      rq_activate_all_grippers(True)
      # end: URCap Program Node
      # begin: URCap Program Node
      #   Source: Robotiq_Grippers, 1.8.13.22852, Robotiq Inc.
      #   Type: Greifer
      $ 271 "Greifer geschlossen (1)"
      if not(gripper_connected[0]):
        popup("Greifer 1 muss verbunden sein, um dieses Programm auszuführen.", "Keine Verbindung", False, True, True)
      end
      if not(rq_is_gripper_activated("1")):
        popup("Greifer 1 ist nicht aktiviert. Wechseln Sie zur Registerkarte Installation > Greifer, um ihn zu aktivieren und das Programm erneut auszuführen.", "Nicht aktiviert", False, True, True)
      end
      rq_set_pos_spd_for(255, 255, 255, "1")
      rq_wait_pos_spe_for_request(255, 255, 255, "1")
      rq_go_to("1")
      rq_wait("1")
      # end: URCap Program Node
      $ 272 "init_qMast≔ False "
      global init_qMast=  False
      $ 273 "Aufruf UserPopups"
      UserPopups()
      $ 274 "Aufruf MachineInputPopUps"
      MachineInputPopUps()
      $ 275 "start_ping≔ True "
      global start_ping=  True
    end
    $ 277 "Switch jobID"
    switch_1 = jobID
    $ 278 "Case 11"
    if (11 == switch_1):
      $ 279 "dest_jobID≔jobArr[1]"
      global dest_jobID=jobArr[1]
      $ 280 "src_dest_p≔qMast.get_loc()"
      global src_dest_p=qMast.get_loc()
      $ 281 "source_p≔src_dest_p[0]"
      global source_p=src_dest_p[0]
      # begin: URCap Program Node
      #   Source: Robotiq_Grippers, 1.8.13.22852, Robotiq Inc.
      #   Type: Greifer
      $ 282 "Greifer geschlossen (1)"
      if not(gripper_connected[0]):
        popup("Greifer 1 muss verbunden sein, um dieses Programm auszuführen.", "Keine Verbindung", False, True, True)
      end
      if not(rq_is_gripper_activated("1")):
        popup("Greifer 1 ist nicht aktiviert. Wechseln Sie zur Registerkarte Installation > Greifer, um ihn zu aktivieren und das Programm erneut auszuführen.", "Nicht aktiviert", False, True, True)
      end
      rq_set_pos_spd_for(255, 255, 255, "1")
      rq_wait_pos_spe_for_request(255, 255, 255, "1")
      rq_go_to("1")
      rq_wait("1")
      # end: URCap Program Node
      $ 283 "FahreAchse"
      $ 284 "stn1_home_p" "breakAfter"
      set_tcp(p[-3.0E-4,2.5E-4,0.1575,0.0,0.0,0.0])
      movej(get_inverse_kin(pose_trans(stn1_plane, pose_trans(p[.053539610991, -.984987293150, -.024848236577, .000189536594, .000276418508, 3.136265531618], stn1_home_p_p)), qnear=stn1_home_p_q), a=3.490658503988659, v=1.0471975511965976, r=0.1)
      $ 285 "FahreAchse"
      $ 286 "stn1_help2_p" "breakAfter"
      set_tcp(p[-3.0E-4,2.5E-4,0.1575,0.0,0.0,0.0])
      movej(get_inverse_kin(pose_trans(stn1_plane, pose_trans(p[.053539610991, -.984987293150, -.024848236577, .000189536594, .000276418508, 3.136265531618], stn1_help2_p_p)), qnear=stn1_help2_p_q), a=1.0471975511965976, v=0.5235987755982988, r=0.05)
      $ 287 "stn1_help_p" "breakAfter"
      set_tcp(p[-3.0E-4,2.5E-4,0.1575,0.0,0.0,0.0])
      movej(get_inverse_kin(pose_trans(stn1_plane, pose_trans(p[.053539610991, -.984987293150, -.024848236577, .000189536594, .000276418508, 3.136265531618], stn1_help_p_p)), qnear=stn1_help_p_q), a=1.0471975511965976, v=0.5235987755982988)
      $ 288 "isStn1Good≔qMast.is_stn1_good()"
      global isStn1Good=qMast.is_stn1_good()
      $ 289 "If isStn1Good ≟  True "
      if (isStn1Good  ==    True  ):
        $ 290 "FahreAchse"
        $ 291 "source_p" "breakAfter"
        set_tcp(p[-3.0E-4,2.5E-4,0.1575,0.0,0.0,0.0])
        movej(pose_trans(stn1_plane, source_p), a=0.8726646259971648, v=0.5235987755982988)
        $ 292 "isStn1Good≔qMast.is_stn1_good()"
        global isStn1Good=qMast.is_stn1_good()
        $ 293 "If isStn1Good ≟  True "
        if (isStn1Good  ==    True  ):
          # begin: URCap Program Node
          #   Source: Robotiq_Grippers, 1.8.13.22852, Robotiq Inc.
          #   Type: Greifer
          $ 294 "Greiferbewegung50% (1)"
          if not(gripper_connected[0]):
            popup("Greifer 1 muss verbunden sein, um dieses Programm auszuführen.", "Keine Verbindung", False, True, True)
          end
          if not(rq_is_gripper_activated("1")):
            popup("Greifer 1 ist nicht aktiviert. Wechseln Sie zur Registerkarte Installation > Greifer, um ihn zu aktivieren und das Programm erneut auszuführen.", "Nicht aktiviert", False, True, True)
          end
          rq_set_pos_spd_for(128, 255, 128, "1")
          rq_wait_pos_spe_for_request(128, 255, 128, "1")
          rq_go_to("1")
          rq_wait("1")
          # end: URCap Program Node
          $ 295 "cur_pose≔pose_trans(pose_inv(stn1_plane), get_actual_tcp_pose())"
          global cur_pose= pose_trans ( pose_inv (stn1_plane),  get_actual_tcp_pose ())
          $ 296 "stn1_pick_p≔pose_trans(cur_pose, p[0,0,stn1_pick_z/1000,0,0,0])"
          global stn1_pick_p= pose_trans (cur_pose, p[0,0,stn1_pick_z/1000,0,0,0])
          $ 297 "FahreLinear"
          $ 298 "stn1_pick_p" "breakAfter"
          set_tcp(p[-3.0E-4,2.5E-4,0.1575,0.0,0.0,0.0])
          movel(pose_trans(stn1_plane, stn1_pick_p), a=0.15, v=0.075)
          $ 299 "isStn1Good≔qMast.is_stn1_good()"
          global isStn1Good=qMast.is_stn1_good()
          $ 300 "If isStn1Good ≟  True "
          if (isStn1Good  ==    True  ):
            # begin: URCap Program Node
            #   Source: Robotiq_Grippers, 1.8.13.22852, Robotiq Inc.
            #   Type: Greifer
            $ 301 "Greifer geschlossen (1)"
            if not(gripper_connected[0]):
              popup("Greifer 1 muss verbunden sein, um dieses Programm auszuführen.", "Keine Verbindung", False, True, True)
            end
            if not(rq_is_gripper_activated("1")):
              popup("Greifer 1 ist nicht aktiviert. Wechseln Sie zur Registerkarte Installation > Greifer, um ihn zu aktivieren und das Programm erneut auszuführen.", "Nicht aktiviert", False, True, True)
            end
            rq_set_pos_spd_for(255, 128, 128, "1")
            rq_wait_pos_spe_for_request(255, 128, 128, "1")
            rq_go_to("1")
            rq_wait("1")
            # end: URCap Program Node
            $ 302 "Warten: 0.2"
            sleep(0.2)
          else:
            $ 303 "Else" "noBreak"
            $ 304 "dest_jobID≔1000"
            global dest_jobID=1000
          end
          $ 305 "FahreAchse"
          $ 306 "source_p" "breakAfter"
          set_tcp(p[-3.0E-4,2.5E-4,0.1575,0.0,0.0,0.0])
          movej(pose_trans(stn1_plane, source_p), a=0.8726646259971648, v=0.5235987755982988)
        else:
          $ 307 "Else" "noBreak"
          $ 308 "dest_jobID≔1000"
          global dest_jobID=1000
        end
      else:
        $ 309 "Else" "noBreak"
        $ 310 "dest_jobID≔1000"
        global dest_jobID=1000
      end
      $ 311 "FahreAchse"
      $ 312 "stn1_help_p" "breakAfter"
      set_tcp(p[-3.0E-4,2.5E-4,0.1575,0.0,0.0,0.0])
      movej(get_inverse_kin(pose_trans(stn1_plane, pose_trans(p[.053539610991, -.984987293150, -.024848236577, .000189536594, .000276418508, 3.136265531618], stn1_help_p_p)), qnear=stn1_help_p_q), a=0.8726646259971648, v=0.5235987755982988, r=0.005)
      $ 313 "stn1_help2_p" "breakAfter"
      set_tcp(p[-3.0E-4,2.5E-4,0.1575,0.0,0.0,0.0])
      movej(get_inverse_kin(pose_trans(stn1_plane, pose_trans(p[.053539610991, -.984987293150, -.024848236577, .000189536594, .000276418508, 3.136265531618], stn1_help2_p_p)), qnear=stn1_help2_p_q), a=0.8726646259971648, v=0.5235987755982988)
      # begin: URCap Program Node
      #   Source: Robotiq_Grippers, 1.8.13.22852, Robotiq Inc.
      #   Type: Griffkontrolle
      $ 314 "Griffkontrolle"
      # begin: URCap Program Node
      #   Source: Robotiq_Grippers, 1.8.13.22852, Robotiq Inc.
      #   Type: Wenn
      $ 315 "Wenn Objekt nicht erkannt          " "noBreak"
      if (not rq_is_object_detected(1)):
        $ 316 "dest_jobID≔1000" "noBreak"
        global dest_jobID=1000
        # end: URCap Program Node
      end
      # end: URCap Program Node
      $ 317 "Switch dest_jobID"
      switch_2 = dest_jobID
      $ 318 "Case 41"
      if (41 == switch_2):
        $ 319 "FahreAchse"
        $ 320 "stn1_home_p" "breakAfter"
        set_tcp(p[-3.0E-4,2.5E-4,0.1575,0.0,0.0,0.0])
        movej(get_inverse_kin(pose_trans(stn1_plane, pose_trans(p[.053539610991, -.984987293150, -.024848236577, .000189536594, .000276418508, 3.136265531618], stn1_home_p_p)), qnear=stn1_home_p_q), a=1.3962634015954636, v=1.0471975511965976, r=0.05)
        $ 321 "FahreAchse"
        $ 322 "stn6_home_p" "breakAfter"
        set_tcp(p[-3.0E-4,2.5E-4,0.1575,0.0,0.0,0.0])
        movej(get_inverse_kin(pose_trans(stn6_plane, pose_trans(p[.776557109756, -.878329076792, .250244777977, -.001605684562, .009314448336, 1.565629725105], stn6_home_p_p)), qnear=stn6_home_p_q), a=3.490658503988659, v=1.0471975511965976, r=0.05)
        $ 323 "stn9_dcap_apr_p" "breakAfter"
        set_tcp(p[-3.0E-4,2.5E-4,0.1575,0.0,0.0,0.0])
        movej(get_inverse_kin(pose_trans(stn6_plane, pose_trans(p[.776557109756, -.878329076792, .250244777977, -.001605684562, .009314448336, 1.565629725105], stn9_dcap_apr_p_p)), qnear=stn9_dcap_apr_p_q), a=3.490658503988659, v=1.0471975511965976)
        $ 324 "Einstellen Decap=Ein"
        set_standard_digital_out(2, True)
        $ 325 "FahreLinear"
        $ 326 "stn9_lv_tb_p" "breakAfter"
        set_tcp(p[-3.0E-4,2.5E-4,0.1575,0.0,0.0,0.0])
        movel(pose_trans(stn6_plane, pose_trans(p[.776557109756, -.878329076792, .250244777977, -.001605684562, .009314448336, 1.565629725105], stn9_lv_tb_p_p)), a=1.2, v=0.25)
        # begin: URCap Program Node
        #   Source: Robotiq_Grippers, 1.8.13.22852, Robotiq Inc.
        #   Type: Greifer
        $ 327 "Greiferbewegung65% (1)"
        if not(gripper_connected[0]):
          popup("Greifer 1 muss verbunden sein, um dieses Programm auszuführen.", "Keine Verbindung", False, True, True)
        end
        if not(rq_is_gripper_activated("1")):
          popup("Greifer 1 ist nicht aktiviert. Wechseln Sie zur Registerkarte Installation > Greifer, um ihn zu aktivieren und das Programm erneut auszuführen.", "Nicht aktiviert", False, True, True)
        end
        rq_set_pos_spd_for(166, 128, 0, "1")
        rq_wait_pos_spe_for_request(166, 128, 0, "1")
        rq_go_to("1")
        rq_wait("1")
        # end: URCap Program Node
        $ 328 "Warten: 0.5"
        sleep(0.5)
        $ 329 "Einstellen Decap=Aus"
        set_standard_digital_out(2, False)
        $ 330 "FahreLinear"
        $ 331 "stn9_hold_cap_p" "breakAfter"
        set_tcp(p[-3.0E-4,2.5E-4,0.1575,0.0,0.0,0.0])
        movel(pose_trans(stn6_plane, pose_trans(p[.776557109756, -.878329076792, .250244777977, -.001605684562, .009314448336, 1.565629725105], stn9_hold_cap_p_p)), a=1.2, v=0.25)
        # begin: URCap Program Node
        #   Source: Robotiq_Grippers, 1.8.13.22852, Robotiq Inc.
        #   Type: Greifer
        $ 332 "Greifer geschlossen (1)"
        if not(gripper_connected[0]):
          popup("Greifer 1 muss verbunden sein, um dieses Programm auszuführen.", "Keine Verbindung", False, True, True)
        end
        if not(rq_is_gripper_activated("1")):
          popup("Greifer 1 ist nicht aktiviert. Wechseln Sie zur Registerkarte Installation > Greifer, um ihn zu aktivieren und das Programm erneut auszuführen.", "Nicht aktiviert", False, True, True)
        end
        rq_set_pos_spd_for(255, 128, 128, "1")
        rq_wait_pos_spe_for_request(255, 128, 128, "1")
        rq_go_to("1")
        rq_wait("1")
        # end: URCap Program Node
        $ 333 "Einstellen Decap=Ein"
        set_standard_digital_out(2, True)
        $ 334 "FahreLinear"
        $ 335 "stn9_dcap_apr_p" "breakAfter"
        set_tcp(p[-3.0E-4,2.5E-4,0.1575,0.0,0.0,0.0])
        movel(pose_trans(stn6_plane, pose_trans(p[.776557109756, -.878329076792, .250244777977, -.001605684562, .009314448336, 1.565629725105], stn9_dcap_apr_p_p)), a=1.2, v=0.25)
        $ 336 "Aufruf stn4_grab_loop"
        stn4_grab_loop()
        $ 337 "dest2_jobID≔qMast.stn4_get_next(stn4_tube_ok)"
        global dest2_jobID=qMast.stn4_get_next(stn4_tube_ok)
        $ 338 "src_dest_p≔qMast.get_loc()"
        global src_dest_p=qMast.get_loc()
        $ 339 "dest_p≔src_dest_p[0]"
        global dest_p=src_dest_p[0]
        $ 340 "Switch dest2_jobID"
        switch_3 = dest2_jobID
        $ 341 "Case 52"
        if (52 == switch_3):
          $ 342 "FahreAchse"
          $ 343 "stn5_stn4_hlp_p" "breakAfter"
          set_tcp(p[-3.0E-4,2.5E-4,0.1575,0.0,0.0,0.0])
          movej(get_inverse_kin(pose_trans(stn6_plane, pose_trans(p[.776557109756, -.878329076792, .250244777977, -.001605684562, .009314448336, 1.565629725105], stn5_stn4_hlp_p_p)), qnear=stn5_stn4_hlp_p_q), a=3.490658503988659, v=1.0471975511965976, r=0.05)
          $ 344 "FahreLinear"
          $ 345 "dest_p" "breakAfter"
          set_tcp(p[-3.0E-4,2.5E-4,0.1575,0.0,0.0,0.0])
          movel(pose_trans(stn5_plane, dest_p), a=1.2, v=0.5)
          $ 346 "cur_pose≔pose_trans(pose_inv(stn5_plane), get_actual_tcp_pose())"
          global cur_pose= pose_trans ( pose_inv (stn5_plane),  get_actual_tcp_pose ())
          $ 347 "stn5_place_z_p≔pose_trans(cur_pose, p[0,0,stn5_place_tb_z/1000,0,0,0])"
          global stn5_place_z_p= pose_trans (cur_pose, p[0,0,stn5_place_tb_z/1000,0,0,0])
          $ 348 "FahreLinear"
          $ 349 "stn5_place_z_p" "breakAfter"
          set_tcp(p[-3.0E-4,2.5E-4,0.1575,0.0,0.0,0.0])
          movel(pose_trans(stn5_plane, stn5_place_z_p), a=0.5, v=0.1)
          # begin: URCap Program Node
          #   Source: Robotiq_Grippers, 1.8.13.22852, Robotiq Inc.
          #   Type: Greifer
          $ 350 "Greiferbewegung50% (1)"
          if not(gripper_connected[0]):
            popup("Greifer 1 muss verbunden sein, um dieses Programm auszuführen.", "Keine Verbindung", False, True, True)
          end
          if not(rq_is_gripper_activated("1")):
            popup("Greifer 1 ist nicht aktiviert. Wechseln Sie zur Registerkarte Installation > Greifer, um ihn zu aktivieren und das Programm erneut auszuführen.", "Nicht aktiviert", False, True, True)
          end
          rq_set_pos_spd_for(127, 255, 255, "1")
          rq_wait_pos_spe_for_request(127, 255, 255, "1")
          rq_go_to("1")
          rq_wait("1")
          # end: URCap Program Node
          $ 351 "dest_p" "breakAfter"
          set_tcp(p[-3.0E-4,2.5E-4,0.1575,0.0,0.0,0.0])
          movel(pose_trans(stn5_plane, dest_p), a=1.2, v=0.25)
          # begin: URCap Program Node
          #   Source: Robotiq_Grippers, 1.8.13.22852, Robotiq Inc.
          #   Type: Greifer
          $ 352 "Greifer geschlossen (1)"
          if not(gripper_connected[0]):
            popup("Greifer 1 muss verbunden sein, um dieses Programm auszuführen.", "Keine Verbindung", False, True, True)
          end
          if not(rq_is_gripper_activated("1")):
            popup("Greifer 1 ist nicht aktiviert. Wechseln Sie zur Registerkarte Installation > Greifer, um ihn zu aktivieren und das Programm erneut auszuführen.", "Nicht aktiviert", False, True, True)
          end
          rq_set_pos_spd_for(255, 255, 255, "1")
          rq_wait_pos_spe_for_request(255, 255, 255, "1")
          rq_go_to("1")
          rq_wait("1")
          # end: URCap Program Node
          $ 353 "FahreAchse"
          $ 354 "stn5_stn4_hlp_p" "breakAfter"
          set_tcp(p[-3.0E-4,2.5E-4,0.1575,0.0,0.0,0.0])
          movej(get_inverse_kin(pose_trans(stn6_plane, pose_trans(p[.776557109756, -.878329076792, .250244777977, -.001605684562, .009314448336, 1.565629725105], stn5_stn4_hlp_p_p)), qnear=stn5_stn4_hlp_p_q), a=1.3962634015954636, v=1.0471975511965976, r=0.05)
          $ 355 "stn6_home_p" "breakAfter"
          set_tcp(p[-3.0E-4,2.5E-4,0.1575,0.0,0.0,0.0])
          movej(get_inverse_kin(pose_trans(stn6_plane, pose_trans(p[.776557109756, -.878329076792, .250244777977, -.001605684562, .009314448336, 1.565629725105], stn6_home_p_p)), qnear=stn6_home_p_q), a=1.3962634015954636, v=1.0471975511965976)
          $ 356 "Aufruf reset_jobs"
          reset_jobs()
        elif (72 == switch_3):
          $ 357 "Case 72"
          $ 358 "FahreAchse"
          $ 359 "stn6_home_p" "breakAfter"
          set_tcp(p[-3.0E-4,2.5E-4,0.1575,0.0,0.0,0.0])
          movej(get_inverse_kin(pose_trans(stn6_plane, pose_trans(p[.776557109756, -.878329076792, .250244777977, -.001605684562, .009314448336, 1.565629725105], stn6_home_p_p)), qnear=stn6_home_p_q), a=3.490658503988659, v=1.0471975511965976, r=0.1)
          $ 360 "FahreAchse"
          $ 361 "stn7_home_p" "breakAfter"
          set_tcp(p[-3.0E-4,2.5E-4,0.1575,0.0,0.0,0.0])
          movej(get_inverse_kin(pose_trans(stn7_plane, pose_trans(p[.109811488584, -1.023382701287, -.166619380160, .003048702642, -.008599620441, 2.442192581404], stn7_home_p_p)), qnear=stn7_home_p_q), a=3.490658503988659, v=1.0471975511965976, r=0.1)
          $ 362 "Aufruf stn7_check_doors"
          stn7_check_doors()
          $ 363 "FahreAchse"
          $ 364 "dest_p" "breakAfter"
          set_tcp(p[-3.0E-4,2.5E-4,0.1575,0.0,0.0,0.0])
          movej(pose_trans(stn7_plane, dest_p), a=3.490658503988659, v=1.0471975511965976)
          $ 365 "cur_pose≔pose_trans(pose_inv(stn7_plane), get_actual_tcp_pose())"
          global cur_pose= pose_trans ( pose_inv (stn7_plane),  get_actual_tcp_pose ())
          $ 366 "stn7_place_p≔pose_trans(cur_pose, p[0,0,stn7_place_z/1000,0,0,0])"
          global stn7_place_p= pose_trans (cur_pose, p[0,0,stn7_place_z/1000,0,0,0])
          $ 367 "FahreLinear"
          $ 368 "stn7_place_p" "breakAfter"
          set_tcp(p[-3.0E-4,2.5E-4,0.1575,0.0,0.0,0.0])
          movel(pose_trans(stn7_plane, stn7_place_p), a=0.15, v=0.075)
          # begin: URCap Program Node
          #   Source: Robotiq_Grippers, 1.8.13.22852, Robotiq Inc.
          #   Type: Greifer
          $ 369 "Greifer offen (1)"
          if not(gripper_connected[0]):
            popup("Greifer 1 muss verbunden sein, um dieses Programm auszuführen.", "Keine Verbindung", False, True, True)
          end
          if not(rq_is_gripper_activated("1")):
            popup("Greifer 1 ist nicht aktiviert. Wechseln Sie zur Registerkarte Installation > Greifer, um ihn zu aktivieren und das Programm erneut auszuführen.", "Nicht aktiviert", False, True, True)
          end
          rq_set_pos_spd_for(0, 255, 255, "1")
          rq_wait_pos_spe_for_request(0, 255, 255, "1")
          rq_go_to("1")
          rq_wait("1")
          # end: URCap Program Node
          $ 370 "FahreLinear"
          $ 371 "dest_p" "breakAfter"
          set_tcp(p[-3.0E-4,2.5E-4,0.1575,0.0,0.0,0.0])
          movel(pose_trans(stn7_plane, dest_p), a=1.2, v=0.25)
          # begin: URCap Program Node
          #   Source: Robotiq_Grippers, 1.8.13.22852, Robotiq Inc.
          #   Type: Greifer
          $ 372 "Greifer geschlossen (1)"
          if not(gripper_connected[0]):
            popup("Greifer 1 muss verbunden sein, um dieses Programm auszuführen.", "Keine Verbindung", False, True, True)
          end
          if not(rq_is_gripper_activated("1")):
            popup("Greifer 1 ist nicht aktiviert. Wechseln Sie zur Registerkarte Installation > Greifer, um ihn zu aktivieren und das Programm erneut auszuführen.", "Nicht aktiviert", False, True, True)
          end
          rq_set_pos_spd_for(255, 255, 255, "1")
          rq_wait_pos_spe_for_request(255, 255, 255, "1")
          rq_go_to("1")
          rq_wait("1")
          # end: URCap Program Node
          $ 373 "FahreAchse"
          $ 374 "stn7_home_p" "breakAfter"
          set_tcp(p[-3.0E-4,2.5E-4,0.1575,0.0,0.0,0.0])
          movej(get_inverse_kin(pose_trans(stn7_plane, pose_trans(p[.109811488584, -1.023382701287, -.166619380160, .003048702642, -.008599620441, 2.442192581404], stn7_home_p_p)), qnear=stn7_home_p_q), a=3.490658503988659, v=1.0471975511965976)
          $ 375 "Aufruf reset_jobs"
          reset_jobs()
        elif (102 == switch_3):
          $ 376 "Case 102"
          $ 377 "FahreAchse"
          $ 378 "stn6_home_p" "breakAfter"
          set_tcp(p[-3.0E-4,2.5E-4,0.1575,0.0,0.0,0.0])
          movej(get_inverse_kin(pose_trans(stn6_plane, pose_trans(p[.776557109756, -.878329076792, .250244777977, -.001605684562, .009314448336, 1.565629725105], stn6_home_p_p)), qnear=stn6_home_p_q), a=3.490658503988659, v=1.0471975511965976, r=0.1)
          $ 379 "stn10_hlp_p" "breakAfter"
          set_tcp(p[-3.0E-4,2.5E-4,0.1575,0.0,0.0,0.0])
          movej(get_inverse_kin(pose_trans(stn6_plane, pose_trans(p[.779413821965, -.869656427631, .149271774994, -.000554336510, .003016566406, 1.568064465904], stn10_hlp_p_p)), qnear=stn10_hlp_p_q), a=3.490658503988659, v=1.0471975511965976)
          $ 380 "FahreLinear"
          $ 381 "dest_p" "breakAfter"
          set_tcp(p[-3.0E-4,2.5E-4,0.1575,0.0,0.0,0.0])
          movel(pose_trans(stn6_plane, dest_p), a=1.2, v=0.5)
          $ 382 "cur_pose≔pose_trans(pose_inv(stn6_plane), get_actual_tcp_pose())"
          global cur_pose= pose_trans ( pose_inv (stn6_plane),  get_actual_tcp_pose ())
          $ 384 "stn10_place_p≔pose_trans(cur_pose, p[0,0,stn10_place_z/1000,0,0,0])"
          global stn10_place_p= pose_trans (cur_pose, p[0,0,stn10_place_z/1000,0,0,0])
          $ 385 "FahreLinear"
          $ 386 "stn10_place_p" "breakAfter"
          set_tcp(p[-3.0E-4,2.5E-4,0.1575,0.0,0.0,0.0])
          movel(pose_trans(stn6_plane, stn10_place_p), a=1.2, v=0.05)
          # begin: URCap Program Node
          #   Source: Robotiq_Grippers, 1.8.13.22852, Robotiq Inc.
          #   Type: Greifer
          $ 387 "Greiferbewegung50% (1)"
          if not(gripper_connected[0]):
            popup("Greifer 1 muss verbunden sein, um dieses Programm auszuführen.", "Keine Verbindung", False, True, True)
          end
          if not(rq_is_gripper_activated("1")):
            popup("Greifer 1 ist nicht aktiviert. Wechseln Sie zur Registerkarte Installation > Greifer, um ihn zu aktivieren und das Programm erneut auszuführen.", "Nicht aktiviert", False, True, True)
          end
          rq_set_pos_spd_for(127, 255, 0, "1")
          rq_wait_pos_spe_for_request(127, 255, 0, "1")
          rq_go_to("1")
          rq_wait("1")
          # end: URCap Program Node
          $ 388 "dest_p" "breakAfter"
          set_tcp(p[-3.0E-4,2.5E-4,0.1575,0.0,0.0,0.0])
          movel(pose_trans(stn6_plane, dest_p), a=1.2, v=0.25)
          # begin: URCap Program Node
          #   Source: Robotiq_Grippers, 1.8.13.22852, Robotiq Inc.
          #   Type: Greifer
          $ 389 "Greifer geschlossen (1)"
          if not(gripper_connected[0]):
            popup("Greifer 1 muss verbunden sein, um dieses Programm auszuführen.", "Keine Verbindung", False, True, True)
          end
          if not(rq_is_gripper_activated("1")):
            popup("Greifer 1 ist nicht aktiviert. Wechseln Sie zur Registerkarte Installation > Greifer, um ihn zu aktivieren und das Programm erneut auszuführen.", "Nicht aktiviert", False, True, True)
          end
          rq_set_pos_spd_for(255, 255, 255, "1")
          rq_wait_pos_spe_for_request(255, 255, 255, "1")
          rq_go_to("1")
          rq_wait("1")
          # end: URCap Program Node
          $ 390 "FahreAchse"
          $ 391 "stn10_hlp_p" "breakAfter"
          set_tcp(p[-3.0E-4,2.5E-4,0.1575,0.0,0.0,0.0])
          movej(get_inverse_kin(pose_trans(stn6_plane, pose_trans(p[.779413821965, -.869656427631, .149271774994, -.000554336510, .003016566406, 1.568064465904], stn10_hlp_p_p)), qnear=stn10_hlp_p_q), a=3.490658503988659, v=1.0471975511965976, r=0.05)
          $ 392 "stn6_home_p" "breakAfter"
          set_tcp(p[-3.0E-4,2.5E-4,0.1575,0.0,0.0,0.0])
          movej(get_inverse_kin(pose_trans(stn6_plane, pose_trans(p[.776557109756, -.878329076792, .250244777977, -.001605684562, .009314448336, 1.565629725105], stn6_home_p_p)), qnear=stn6_home_p_q), a=3.490658503988659, v=1.0471975511965976)
          $ 393 "Aufruf reset_jobs"
          reset_jobs()
        elif (152 == switch_3):
          $ 394 "Case 152"
          $ 395 "FahreAchse"
          $ 396 "stn11_hlp_p" "breakAfter"
          set_tcp(p[-3.0E-4,2.5E-4,0.1575,0.0,0.0,0.0])
          movej(get_inverse_kin(pose_trans(stn6_plane, pose_trans(p[.776557109756, -.878329076792, .250244777977, -.001605684562, .009314448336, 1.565629725105], stn11_hlp_p_p)), qnear=stn11_hlp_p_q), a=2.0943951023931953, v=1.0471975511965976, r=0.05)
          $ 397 "stn15_home_p" "breakAfter"
          set_tcp(p[-3.0E-4,2.5E-4,0.1575,0.0,0.0,0.0])
          movej(get_inverse_kin(pose_trans(stn6_plane, pose_trans(p[.776557109756, -.878329076792, .250244777977, -.001605684562, .009314448336, 1.565629725105], stn15_home_p_p)), qnear=stn15_home_p_q), a=2.0943951023931953, v=1.0471975511965976, r=0.01)
          $ 398 "dest_p" "breakAfter"
          set_tcp(p[-3.0E-4,2.5E-4,0.1575,0.0,0.0,0.0])
          movej(pose_trans(stn6_plane, dest_p), a=2.0943951023931953, v=1.0471975511965976)
          $ 399 "cur_pose≔pose_trans(pose_inv(stn6_plane), get_actual_tcp_pose())"
          global cur_pose= pose_trans ( pose_inv (stn6_plane),  get_actual_tcp_pose ())
          $ 400 "stn15_place_z_p≔pose_trans(cur_pose, p[0,0,stn15_place_z/1000,0,0,0])"
          global stn15_place_z_p= pose_trans (cur_pose, p[0,0,stn15_place_z/1000,0,0,0])
          $ 401 "FahreLinear"
          $ 402 "stn15_place_z_p" "breakAfter"
          set_tcp(p[-3.0E-4,2.5E-4,0.1575,0.0,0.0,0.0])
          movel(pose_trans(stn6_plane, stn15_place_z_p), a=0.5, v=0.1)
          # begin: URCap Program Node
          #   Source: Robotiq_Grippers, 1.8.13.22852, Robotiq Inc.
          #   Type: Greifer
          $ 403 "Greiferbewegung50% (1)"
          if not(gripper_connected[0]):
            popup("Greifer 1 muss verbunden sein, um dieses Programm auszuführen.", "Keine Verbindung", False, True, True)
          end
          if not(rq_is_gripper_activated("1")):
            popup("Greifer 1 ist nicht aktiviert. Wechseln Sie zur Registerkarte Installation > Greifer, um ihn zu aktivieren und das Programm erneut auszuführen.", "Nicht aktiviert", False, True, True)
          end
          rq_set_pos_spd_for(128, 255, 255, "1")
          rq_wait_pos_spe_for_request(128, 255, 255, "1")
          rq_go_to("1")
          rq_wait("1")
          # end: URCap Program Node
          $ 404 "dest_p" "breakAfter"
          set_tcp(p[-3.0E-4,2.5E-4,0.1575,0.0,0.0,0.0])
          movel(pose_trans(stn6_plane, dest_p), a=0.5, v=0.1)
          # begin: URCap Program Node
          #   Source: Robotiq_Grippers, 1.8.13.22852, Robotiq Inc.
          #   Type: Greifer
          $ 405 "Greifer geschlossen (1)"
          if not(gripper_connected[0]):
            popup("Greifer 1 muss verbunden sein, um dieses Programm auszuführen.", "Keine Verbindung", False, True, True)
          end
          if not(rq_is_gripper_activated("1")):
            popup("Greifer 1 ist nicht aktiviert. Wechseln Sie zur Registerkarte Installation > Greifer, um ihn zu aktivieren und das Programm erneut auszuführen.", "Nicht aktiviert", False, True, True)
          end
          rq_set_pos_spd_for(255, 255, 255, "1")
          rq_wait_pos_spe_for_request(255, 255, 255, "1")
          rq_go_to("1")
          rq_wait("1")
          # end: URCap Program Node
          $ 406 "FahreAchse"
          $ 407 "stn15_home_p" "breakAfter"
          set_tcp(p[-3.0E-4,2.5E-4,0.1575,0.0,0.0,0.0])
          movej(get_inverse_kin(pose_trans(stn6_plane, pose_trans(p[.776557109756, -.878329076792, .250244777977, -.001605684562, .009314448336, 1.565629725105], stn15_home_p_p)), qnear=stn15_home_p_q), a=2.0943951023931953, v=1.0471975511965976, r=0.05)
          $ 408 "FahreAchse"
          $ 409 "stn1_home_p" "breakAfter"
          set_tcp(p[-3.0E-4,2.5E-4,0.1575,0.0,0.0,0.0])
          movej(get_inverse_kin(pose_trans(stn1_plane, pose_trans(p[.053539610991, -.984987293150, -.024848236577, .000189536594, .000276418508, 3.136265531618], stn1_home_p_p)), qnear=stn1_home_p_q), a=2.0943951023931953, v=1.0471975511965976)
          $ 410 "Aufruf reset_jobs"
          reset_jobs()
        end
      elif (1000 == switch_2):
        $ 411 "Case 1000"
        $ 412 "FahreAchse"
        $ 413 "stn1_home_p" "breakAfter"
        set_tcp(p[-3.0E-4,2.5E-4,0.1575,0.0,0.0,0.0])
        movej(get_inverse_kin(pose_trans(stn1_plane, pose_trans(p[.053539610991, -.984987293150, -.024848236577, .000189536594, .000276418508, 3.136265531618], stn1_home_p_p)), qnear=stn1_home_p_q), a=3.490658503988659, v=1.0471975511965976)
        # begin: URCap Program Node
        #   Source: Robotiq_Grippers, 1.8.13.22852, Robotiq Inc.
        #   Type: Greifer
        $ 414 "Greifer geschlossen (1)"
        if not(gripper_connected[0]):
          popup("Greifer 1 muss verbunden sein, um dieses Programm auszuführen.", "Keine Verbindung", False, True, True)
        end
        if not(rq_is_gripper_activated("1")):
          popup("Greifer 1 ist nicht aktiviert. Wechseln Sie zur Registerkarte Installation > Greifer, um ihn zu aktivieren und das Programm erneut auszuführen.", "Nicht aktiviert", False, True, True)
        end
        rq_set_pos_spd_for(255, 128, 128, "1")
        rq_wait_pos_spe_for_request(255, 128, 128, "1")
        rq_go_to("1")
        rq_wait("1")
        # end: URCap Program Node
        $ 415 "Aufruf reset_jobs"
        reset_jobs()
      end
    elif (21 == switch_1):
      $ 416 "Case 21"
      $ 417 "dest_jobID≔jobArr[1]"
      global dest_jobID=jobArr[1]
      $ 418 "src_dest_p≔qMast.get_loc()"
      global src_dest_p=qMast.get_loc()
      $ 419 "source_p≔src_dest_p[0]"
      global source_p=src_dest_p[0]
      $ 420 "Switch dest_jobID"
      switch_2 = dest_jobID
      $ 421 "Case 142"
      if (142 == switch_2):
        $ 422 "FahreAchse"
        $ 423 "stn2_home_p" "breakAfter"
        set_tcp(p[-3.0E-4,2.5E-4,0.1575,0.0,0.0,0.0])
        movej(get_inverse_kin(pose_trans(stn2_plane, pose_trans(p[.137500819741, -.686313800478, .149495066037, -.008721928164, .022313263547, 3.131433712319], stn2_home_p_p)), qnear=stn2_home_p_q), a=1.3962634015954636, v=1.0471975511965976)
        $ 424 "source_p" "breakAfter"
        set_tcp(p[-3.0E-4,2.5E-4,0.1575,0.0,0.0,0.0])
        movej(pose_trans(stn2_plane, source_p), a=1.3962634015954636, v=1.0471975511965976)
        # begin: URCap Program Node
        #   Source: Robotiq_Grippers, 1.8.13.22852, Robotiq Inc.
        #   Type: Greifer
        $ 425 "Greiferbewegung35% (1)"
        if not(gripper_connected[0]):
          popup("Greifer 1 muss verbunden sein, um dieses Programm auszuführen.", "Keine Verbindung", False, True, True)
        end
        if not(rq_is_gripper_activated("1")):
          popup("Greifer 1 ist nicht aktiviert. Wechseln Sie zur Registerkarte Installation > Greifer, um ihn zu aktivieren und das Programm erneut auszuführen.", "Nicht aktiviert", False, True, True)
        end
        rq_set_pos_spd_for(89, 255, 255, "1")
        rq_wait_pos_spe_for_request(89, 255, 255, "1")
        rq_go_to("1")
        rq_wait("1")
        # end: URCap Program Node
        $ 426 "cur_pose≔pose_trans(pose_inv(stn2_plane), get_actual_tcp_pose())"
        global cur_pose= pose_trans ( pose_inv (stn2_plane),  get_actual_tcp_pose ())
        $ 427 "stn2_pick_z_p≔pose_trans(cur_pose, p[0,0,stn2_pk_rk_z/1000,0,0,0])"
        global stn2_pick_z_p= pose_trans (cur_pose, p[0,0,stn2_pk_rk_z/1000,0,0,0])
        $ 428 "FahreLinear"
        $ 429 "stn2_pick_z_p" "breakAfter"
        set_tcp(p[-3.0E-4,2.5E-4,0.1575,0.0,0.0,0.0])
        movel(pose_trans(stn2_plane, stn2_pick_z_p), a=0.5, v=0.1)
        $ 430 "cur_pose≔pose_trans(pose_inv(stn2_plane), get_actual_tcp_pose())"
        global cur_pose= pose_trans ( pose_inv (stn2_plane),  get_actual_tcp_pose ())
        $ 431 "stn2_rk_chk_y_p≔pose_trans(cur_pose, p[0,stn2_rk_chk_y/1000,0,0,0,0])"
        global stn2_rk_chk_y_p= pose_trans (cur_pose, p[0,stn2_rk_chk_y/1000,0,0,0,0])
        $ 432 "FahreLinear"
        $ 433 "stn2_rk_chk_y_p" "breakAfter"
        set_tcp(p[-3.0E-4,2.5E-4,0.1575,0.0,0.0,0.0])
        movel(pose_trans(stn2_plane, stn2_rk_chk_y_p), a=0.5, v=0.1)
        $ 434 "stn14_angle≔0"
        global stn14_angle=0
        $ 435 "stn2_rack_yes≔ False "
        global stn2_rack_yes=  False
        # begin: URCap Program Node
        #   Source: Robotiq_Grippers, 1.8.13.22852, Robotiq Inc.
        #   Type: Greifer
        $ 436 "Greifer geschlossen (1)"
        if not(gripper_connected[0]):
          popup("Greifer 1 muss verbunden sein, um dieses Programm auszuführen.", "Keine Verbindung", False, True, True)
        end
        if not(rq_is_gripper_activated("1")):
          popup("Greifer 1 ist nicht aktiviert. Wechseln Sie zur Registerkarte Installation > Greifer, um ihn zu aktivieren und das Programm erneut auszuführen.", "Nicht aktiviert", False, True, True)
        end
        rq_set_pos_spd_for(255, 0, 0, "1")
        rq_wait_pos_spe_for_request(255, 0, 0, "1")
        rq_go_to("1")
        rq_wait("1")
        # end: URCap Program Node
        $ 437 "gripper_pos≔rq_current_pos_norm()"
        global gripper_pos=rq_current_pos_norm()
        $ 438 "If gripper_pos ≤ 65 and gripper_pos ≥ 57"
        if (gripper_pos  <=  65  and  gripper_pos  >=  57):
          $ 439 "stn2_rack_yes≔ True "
          global stn2_rack_yes=  True
          $ 440 "stn14_angle≔180"
          global stn14_angle=180
        else:
          $ 441 "ElseIf gripper_pos > 65  and gripper_pos ≤ 90"
          if (gripper_pos > 65   and  gripper_pos  <=  90):
            $ 442 "stn2_rack_yes≔ True "
            global stn2_rack_yes=  True
          else:
            $ 443 "Else" "noBreak"
            $ 444 "stn2_rack_yes≔ False "
            global stn2_rack_yes=  False
          end
        end
        # begin: URCap Program Node
        #   Source: Robotiq_Grippers, 1.8.13.22852, Robotiq Inc.
        #   Type: Greifer
        $ 445 "Greiferbewegung35% (1)"
        if not(gripper_connected[0]):
          popup("Greifer 1 muss verbunden sein, um dieses Programm auszuführen.", "Keine Verbindung", False, True, True)
        end
        if not(rq_is_gripper_activated("1")):
          popup("Greifer 1 ist nicht aktiviert. Wechseln Sie zur Registerkarte Installation > Greifer, um ihn zu aktivieren und das Programm erneut auszuführen.", "Nicht aktiviert", False, True, True)
        end
        rq_set_pos_spd_for(89, 255, 255, "1")
        rq_wait_pos_spe_for_request(89, 255, 255, "1")
        rq_go_to("1")
        rq_wait("1")
        # end: URCap Program Node
        $ 446 "FahreLinear"
        $ 447 "stn2_pick_z_p" "breakAfter"
        set_tcp(p[-3.0E-4,2.5E-4,0.1575,0.0,0.0,0.0])
        movel(pose_trans(stn2_plane, stn2_pick_z_p), a=1.2, v=0.25)
        $ 448 "If stn2_rack_yes ≟  True "
        if (stn2_rack_yes  ==    True  ):
          # begin: URCap Program Node
          #   Source: Robotiq_Grippers, 1.8.13.22852, Robotiq Inc.
          #   Type: Greifer
          $ 449 "Greifer geschlossen (1)"
          if not(gripper_connected[0]):
            popup("Greifer 1 muss verbunden sein, um dieses Programm auszuführen.", "Keine Verbindung", False, True, True)
          end
          if not(rq_is_gripper_activated("1")):
            popup("Greifer 1 ist nicht aktiviert. Wechseln Sie zur Registerkarte Installation > Greifer, um ihn zu aktivieren und das Programm erneut auszuführen.", "Nicht aktiviert", False, True, True)
          end
          rq_set_pos_spd_for(255, 128, 255, "1")
          rq_wait_pos_spe_for_request(255, 128, 255, "1")
          rq_go_to("1")
          rq_wait("1")
          # end: URCap Program Node
          $ 450 "FahreLinear"
          $ 451 "source_p" "breakAfter"
          set_tcp(p[-3.0E-4,2.5E-4,0.1575,0.0,0.0,0.0])
          movel(pose_trans(stn2_plane, source_p), a=0.5, v=0.1)
          $ 452 "FahreAchse"
          $ 453 "stn2_home_p" "breakAfter"
          set_tcp(p[-3.0E-4,2.5E-4,0.1575,0.0,0.0,0.0])
          movej(get_inverse_kin(pose_trans(stn2_plane, pose_trans(p[.137500819741, -.686313800478, .149495066037, -.008721928164, .022313263547, 3.131433712319], stn2_home_p_p)), qnear=stn2_home_p_q), a=1.3962634015954636, v=1.0471975511965976)
          $ 454 "FahreAchse"
          $ 455 "stn6_home_p" "breakAfter"
          set_tcp(p[-3.0E-4,2.5E-4,0.1575,0.0,0.0,0.0])
          movej(get_inverse_kin(pose_trans(stn6_plane, pose_trans(p[.776557109756, -.878329076792, .250244777977, -.001605684562, .009314448336, 1.565629725105], stn6_home_p_p)), qnear=stn6_home_p_q), a=1.3962634015954636, v=1.0471975511965976, r=0.1)
          $ 456 "stn14_pl_rk_h_p" "breakAfter"
          set_tcp(p[-3.0E-4,2.5E-4,0.1575,0.0,0.0,0.0])
          movej(get_inverse_kin(pose_trans(stn6_plane, pose_trans(p[.776557109756, -.878329076792, .250244777977, -.001605684562, .009314448336, 1.565629725105], stn14_pl_rk_h_p_p)), qnear=stn14_pl_rk_h_p_q), a=1.3962634015954636, v=1.0471975511965976, r=0.05)
          $ 457 "stn14_pl_rk_p" "breakAfter"
          set_tcp(p[-3.0E-4,2.5E-4,0.1575,0.0,0.0,0.0])
          movej(get_inverse_kin(pose_trans(stn6_plane, pose_trans(p[.776557109756, -.878329076792, .250244777977, -.001605684562, .009314448336, 1.565629725105], stn14_pl_rk_p_p)), qnear=stn14_pl_rk_p_q), a=1.3962634015954636, v=1.0471975511965976)
          $ 458 "If stn14_angle ≟ 180"
          if (stn14_angle  ==  180):
            $ 459 "FahreAchse"
            $ 460 "stn14_plrk_rt_p" "breakAfter"
            set_tcp(p[-3.0E-4,2.5E-4,0.1575,0.0,0.0,0.0])
            movej(get_inverse_kin(pose_trans(stn6_plane, pose_trans(p[.776557109756, -.878329076792, .250244777977, -.001605684562, .009314448336, 1.565629725105], stn14_plrk_rt_p_p)), qnear=stn14_plrk_rt_p_q), a=13.962634015954636, v=3.141592653589793)
            $ 461 "FahreLinear"
            $ 462 "cur_pose≔pose_trans(pose_inv(stn6_plane), get_actual_tcp_pose())"
            global cur_pose= pose_trans ( pose_inv (stn6_plane),  get_actual_tcp_pose ())
            $ 463 "stn14_pl_rk_z_p≔pose_trans(cur_pose, p[0,0,stn14_pl_rk_z/1000,0,0,0])"
            global stn14_pl_rk_z_p= pose_trans (cur_pose, p[0,0,stn14_pl_rk_z/1000,0,0,0])
            $ 464 "stn14_pl_rk_z_p" "breakAfter"
            set_tcp(p[-3.0E-4,2.5E-4,0.1575,0.0,0.0,0.0])
            movel(pose_trans(stn6_plane, stn14_pl_rk_z_p), a=0.5, v=0.05)
            # begin: URCap Program Node
            #   Source: Robotiq_Grippers, 1.8.13.22852, Robotiq Inc.
            #   Type: Greifer
            $ 465 "Greiferbewegung35% (1)"
            if not(gripper_connected[0]):
              popup("Greifer 1 muss verbunden sein, um dieses Programm auszuführen.", "Keine Verbindung", False, True, True)
            end
            if not(rq_is_gripper_activated("1")):
              popup("Greifer 1 ist nicht aktiviert. Wechseln Sie zur Registerkarte Installation > Greifer, um ihn zu aktivieren und das Programm erneut auszuführen.", "Nicht aktiviert", False, True, True)
            end
            rq_set_pos_spd_for(89, 255, 255, "1")
            rq_wait_pos_spe_for_request(89, 255, 255, "1")
            rq_go_to("1")
            rq_wait("1")
            # end: URCap Program Node
            $ 466 "stn14_plrk_rt_p" "breakAfter"
            set_tcp(p[-3.0E-4,2.5E-4,0.1575,0.0,0.0,0.0])
            movel(pose_trans(stn6_plane, pose_trans(p[.776557109756, -.878329076792, .250244777977, -.001605684562, .009314448336, 1.565629725105], stn14_plrk_rt_p_p)), a=0.6, v=0.1)
            # begin: URCap Program Node
            #   Source: Robotiq_Grippers, 1.8.13.22852, Robotiq Inc.
            #   Type: Greifer
            $ 467 "Greifer geschlossen (1)"
            if not(gripper_connected[0]):
              popup("Greifer 1 muss verbunden sein, um dieses Programm auszuführen.", "Keine Verbindung", False, True, True)
            end
            if not(rq_is_gripper_activated("1")):
              popup("Greifer 1 ist nicht aktiviert. Wechseln Sie zur Registerkarte Installation > Greifer, um ihn zu aktivieren und das Programm erneut auszuführen.", "Nicht aktiviert", False, True, True)
            end
            rq_set_pos_spd_for(255, 255, 255, "1")
            rq_wait_pos_spe_for_request(255, 255, 255, "1")
            rq_go_to("1")
            rq_wait("1")
            # end: URCap Program Node
          else:
            $ 468 "Else" "noBreak"
            $ 469 "FahreLinear"
            $ 470 "cur_pose≔pose_trans(pose_inv(stn6_plane), get_actual_tcp_pose())"
            global cur_pose= pose_trans ( pose_inv (stn6_plane),  get_actual_tcp_pose ())
            $ 471 "stn14_pl_rk_z_p≔pose_trans(cur_pose, p[0,0,stn14_pl_rk_z/1000,0,0,0])"
            global stn14_pl_rk_z_p= pose_trans (cur_pose, p[0,0,stn14_pl_rk_z/1000,0,0,0])
            $ 472 "stn14_pl_rk_z_p" "breakAfter"
            set_tcp(p[-3.0E-4,2.5E-4,0.1575,0.0,0.0,0.0])
            movel(pose_trans(stn6_plane, stn14_pl_rk_z_p), a=0.5, v=0.05)
            # begin: URCap Program Node
            #   Source: Robotiq_Grippers, 1.8.13.22852, Robotiq Inc.
            #   Type: Greifer
            $ 473 "Greiferbewegung35% (1)"
            if not(gripper_connected[0]):
              popup("Greifer 1 muss verbunden sein, um dieses Programm auszuführen.", "Keine Verbindung", False, True, True)
            end
            if not(rq_is_gripper_activated("1")):
              popup("Greifer 1 ist nicht aktiviert. Wechseln Sie zur Registerkarte Installation > Greifer, um ihn zu aktivieren und das Programm erneut auszuführen.", "Nicht aktiviert", False, True, True)
            end
            rq_set_pos_spd_for(89, 255, 255, "1")
            rq_wait_pos_spe_for_request(89, 255, 255, "1")
            rq_go_to("1")
            rq_wait("1")
            # end: URCap Program Node
            $ 474 "stn14_pl_rk_p" "breakAfter"
            set_tcp(p[-3.0E-4,2.5E-4,0.1575,0.0,0.0,0.0])
            movel(pose_trans(stn6_plane, pose_trans(p[.776557109756, -.878329076792, .250244777977, -.001605684562, .009314448336, 1.565629725105], stn14_pl_rk_p_p)), a=0.5, v=0.1)
            # begin: URCap Program Node
            #   Source: Robotiq_Grippers, 1.8.13.22852, Robotiq Inc.
            #   Type: Greifer
            $ 475 "Greifer geschlossen (1)"
            if not(gripper_connected[0]):
              popup("Greifer 1 muss verbunden sein, um dieses Programm auszuführen.", "Keine Verbindung", False, True, True)
            end
            if not(rq_is_gripper_activated("1")):
              popup("Greifer 1 ist nicht aktiviert. Wechseln Sie zur Registerkarte Installation > Greifer, um ihn zu aktivieren und das Programm erneut auszuführen.", "Nicht aktiviert", False, True, True)
            end
            rq_set_pos_spd_for(255, 255, 255, "1")
            rq_wait_pos_spe_for_request(255, 255, 255, "1")
            rq_go_to("1")
            rq_wait("1")
            # end: URCap Program Node
          end
          $ 476 "FahreAchse"
          $ 477 "stn6_home_p" "breakAfter"
          set_tcp(p[-3.0E-4,2.5E-4,0.1575,0.0,0.0,0.0])
          movej(get_inverse_kin(pose_trans(stn6_plane, pose_trans(p[.776557109756, -.878329076792, .250244777977, -.001605684562, .009314448336, 1.565629725105], stn6_home_p_p)), qnear=stn6_home_p_q), a=1.3962634015954636, v=1.0471975511965976)
          $ 478 "qMast.stn14_fill_holder()"
          qMast.stn14_fill_holder()
        else:
          $ 479 "Else" "noBreak"
          $ 480 "FahreLinear"
          $ 481 "source_p" "breakAfter"
          set_tcp(p[-3.0E-4,2.5E-4,0.1575,0.0,0.0,0.0])
          movel(pose_trans(stn2_plane, source_p), a=1.2, v=0.25)
          $ 482 "FahreAchse"
          $ 483 "stn2_home_p" "breakAfter"
          set_tcp(p[-3.0E-4,2.5E-4,0.1575,0.0,0.0,0.0])
          movej(get_inverse_kin(pose_trans(stn2_plane, pose_trans(p[.137500819741, -.686313800478, .149495066037, -.008721928164, .022313263547, 3.131433712319], stn2_home_p_p)), qnear=stn2_home_p_q), a=1.3962634015954636, v=1.0471975511965976)
        end
        $ 484 "Aufruf reset_jobs"
        reset_jobs()
      end
    elif (23 == switch_1):
      $ 485 "Case 23"
      $ 486 "Aufruf stn2_door1_close"
      stn2_door1_close()
      $ 487 "Aufruf stn2_door1_open"
      stn2_door1_open()
      $ 488 "Aufruf reset_jobs"
      reset_jobs()
    elif (24 == switch_1):
      $ 489 "Case 24"
      $ 490 "Aufruf stn2_door1_close"
      stn2_door1_close()
      $ 491 "FahreAchse"
      $ 492 "stn2_home_p" "breakAfter"
      set_tcp(p[-3.0E-4,2.5E-4,0.1575,0.0,0.0,0.0])
      movej(get_inverse_kin(pose_trans(stn2_plane, pose_trans(p[.137500819741, -.686313800478, .149495066037, -.008721928164, .022313263547, 3.131433712319], stn2_home_p_p)), qnear=stn2_home_p_q), a=1.3962634015954636, v=1.0471975511965976)
      $ 493 "Aufruf reset_jobs"
      reset_jobs()
    elif (25 == switch_1):
      $ 494 "Case 25"
      $ 495 "Aufruf stn2_door2_close"
      stn2_door2_close()
      $ 496 "Aufruf stn2_door2_open"
      stn2_door2_open()
      $ 497 "Aufruf reset_jobs"
      reset_jobs()
    elif (26 == switch_1):
      $ 498 "Case 26"
      $ 499 "Aufruf stn2_door2_close"
      stn2_door2_close()
      $ 500 "FahreAchse"
      $ 501 "stn2_home_p" "breakAfter"
      set_tcp(p[-3.0E-4,2.5E-4,0.1575,0.0,0.0,0.0])
      movej(get_inverse_kin(pose_trans(stn2_plane, pose_trans(p[.137500819741, -.686313800478, .149495066037, -.008721928164, .022313263547, 3.131433712319], stn2_home_p_p)), qnear=stn2_home_p_q), a=1.3962634015954636, v=1.0471975511965976)
      $ 502 "Aufruf reset_jobs"
      reset_jobs()
    elif (27 == switch_1):
      $ 503 "Case 27"
      $ 504 "Aufruf stn2_door3_close"
      stn2_door3_close()
      $ 505 "Aufruf stn2_door3_open"
      stn2_door3_open()
      $ 506 "Aufruf reset_jobs"
      reset_jobs()
    elif (28 == switch_1):
      $ 507 "Case 28"
      $ 508 "Aufruf stn2_door3_close"
      stn2_door3_close()
      $ 509 "FahreAchse"
      $ 510 "stn2_home_p" "breakAfter"
      set_tcp(p[-3.0E-4,2.5E-4,0.1575,0.0,0.0,0.0])
      movej(get_inverse_kin(pose_trans(stn2_plane, pose_trans(p[.137500819741, -.686313800478, .149495066037, -.008721928164, .022313263547, 3.131433712319], stn2_home_p_p)), qnear=stn2_home_p_q), a=1.3962634015954636, v=1.0471975511965976)
      $ 511 "Aufruf reset_jobs"
      reset_jobs()
    elif (29 == switch_1):
      $ 512 "Case 29"
      $ 513 "FahreAchse"
      $ 514 "stn2_home_p" "breakAfter"
      set_tcp(p[-3.0E-4,2.5E-4,0.1575,0.0,0.0,0.0])
      movej(get_inverse_kin(pose_trans(stn2_plane, pose_trans(p[.137500819741, -.686313800478, .149495066037, -.008721928164, .022313263547, 3.131433712319], stn2_home_p_p)), qnear=stn2_home_p_q), a=1.3962634015954636, v=1.0471975511965976)
      $ 515 "FahreAchse"
      $ 516 "stn1_home_p" "breakAfter"
      set_tcp(p[-3.0E-4,2.5E-4,0.1575,0.0,0.0,0.0])
      movej(get_inverse_kin(pose_trans(stn1_plane, pose_trans(p[.053539610991, -.984987293150, -.024848236577, .000189536594, .000276418508, 3.136265531618], stn1_home_p_p)), qnear=stn1_home_p_q), a=1.3962634015954636, v=1.0471975511965976)
      $ 517 "home_p" "breakAfter"
      set_tcp(p[-3.0E-4,2.5E-4,0.1575,0.0,0.0,0.0])
      movej(get_inverse_kin(pose_trans(stn1_plane, pose_trans(p[.053539610991, -.984987293150, -.024848236577, .000189536594, .000276418508, 3.136265531618], home_p_p)), qnear=home_p_q), a=1.3962634015954636, v=1.0471975511965976)
      $ 518 "Meldung: Alle Cobas Racks benutzen"
      popup("Alle Cobas Racks benutzen", "Fehler", False, True, blocking=False)
      halt
      $ 519 "Aufruf reset_jobs"
      reset_jobs()
    elif (30 == switch_1):
      $ 520 "Case 30"
      $ 521 "If Test ≟  True "
      if (Test  ==    True  ):
        $ 522 "qMast.set_init_alarm(3)"
        qMast.set_init_alarm(3)
      else:
        $ 523 "Else" "noBreak"
        $ 524 "Aufruf stn3_init_stndby"
        stn3_init_stndby()
        $ 525 "qMast.set_init_alarm(3)"
        qMast.set_init_alarm(3)
        $ 526 "FahreAchse"
        $ 527 "stn3_home_p" "breakAfter"
        set_tcp(p[-3.0E-4,2.5E-4,0.1575,0.0,0.0,0.0])
        movej(get_inverse_kin(pose_trans(stn3_plane, pose_trans(p[.103513391500, -.760903866624, .250613495596, .000363058783, .000522680433, -.002816727210], stn3_home_p_p)), qnear=stn3_home_p_q), a=1.3962634015954636, v=1.0471975511965976)
      end
      $ 528 "Aufruf reset_jobs"
      reset_jobs()
    elif (31 == switch_1):
      $ 529 "Case 31"
      $ 530 "dest_jobID≔jobArr[1]"
      global dest_jobID=jobArr[1]
      $ 531 "src_dest_p≔qMast.get_loc()"
      global src_dest_p=qMast.get_loc()
      $ 532 "source_p≔src_dest_p[0]"
      global source_p=src_dest_p[0]
      $ 533 "FahreAchse"
      $ 534 "stn3_home_p" "breakAfter"
      set_tcp(p[-3.0E-4,2.5E-4,0.1575,0.0,0.0,0.0])
      movej(get_inverse_kin(pose_trans(stn3_plane, pose_trans(p[.103513391500, -.760903866624, .250613495596, .000363058783, .000522680433, -.002816727210], stn3_home_p_p)), qnear=stn3_home_p_q), a=1.3962634015954636, v=1.0471975511965976, r=0.1)
      $ 535 "stn3_top_hlp_p" "breakAfter"
      set_tcp(p[-3.0E-4,2.5E-4,0.1575,0.0,0.0,0.0])
      movej(get_inverse_kin(pose_trans(stn3_plane, pose_trans(p[.103513391500, -.760903866624, .250613495596, .000363058783, .000522680433, -.002816727210], stn3_top_hlp_p_p)), qnear=stn3_top_hlp_p_q), a=2.792526803190927, v=1.7453292519943295, r=0.02)
      $ 536 "source_p" "breakAfter"
      set_tcp(p[-3.0E-4,2.5E-4,0.1575,0.0,0.0,0.0])
      movej(pose_trans(stn3_plane, source_p), a=1.3962634015954636, v=1.0471975511965976)
      # begin: URCap Program Node
      #   Source: Robotiq_Grippers, 1.8.13.22852, Robotiq Inc.
      #   Type: Greifer
      $ 537 "Greiferbewegung50% (1)"
      if not(gripper_connected[0]):
        popup("Greifer 1 muss verbunden sein, um dieses Programm auszuführen.", "Keine Verbindung", False, True, True)
      end
      if not(rq_is_gripper_activated("1")):
        popup("Greifer 1 ist nicht aktiviert. Wechseln Sie zur Registerkarte Installation > Greifer, um ihn zu aktivieren und das Programm erneut auszuführen.", "Nicht aktiviert", False, True, True)
      end
      rq_set_pos_spd_for(128, 128, 128, "1")
      rq_wait_pos_spe_for_request(128, 128, 128, "1")
      rq_go_to("1")
      rq_wait("1")
      # end: URCap Program Node
      $ 538 "cur_pose≔pose_trans(pose_inv(stn3_plane), get_actual_tcp_pose())"
      global cur_pose= pose_trans ( pose_inv (stn3_plane),  get_actual_tcp_pose ())
      $ 539 "stn3_pick_p≔pose_trans(cur_pose, p[0,0,stn3_pick_z/1000,0,0,0])"
      global stn3_pick_p= pose_trans (cur_pose, p[0,0,stn3_pick_z/1000,0,0,0])
      $ 540 "FahreLinear"
      $ 541 "stn3_pick_p" "breakAfter"
      set_tcp(p[-3.0E-4,2.5E-4,0.1575,0.0,0.0,0.0])
      movel(pose_trans(stn3_plane, stn3_pick_p), a=0.2, v=0.05)
      # begin: URCap Program Node
      #   Source: Robotiq_Grippers, 1.8.13.22852, Robotiq Inc.
      #   Type: Greifer
      $ 542 "Greifer geschlossen (1)"
      if not(gripper_connected[0]):
        popup("Greifer 1 muss verbunden sein, um dieses Programm auszuführen.", "Keine Verbindung", False, True, True)
      end
      if not(rq_is_gripper_activated("1")):
        popup("Greifer 1 ist nicht aktiviert. Wechseln Sie zur Registerkarte Installation > Greifer, um ihn zu aktivieren und das Programm erneut auszuführen.", "Nicht aktiviert", False, True, True)
      end
      rq_set_pos_spd_for(255, 128, 128, "1")
      rq_wait_pos_spe_for_request(255, 128, 128, "1")
      rq_go_to("1")
      rq_wait("1")
      # end: URCap Program Node
      $ 543 "source_p" "breakAfter"
      set_tcp(p[-3.0E-4,2.5E-4,0.1575,0.0,0.0,0.0])
      movel(pose_trans(stn3_plane, source_p), a=0.2, v=0.05)
      $ 544 "dest_p≔src_dest_p[1]"
      global dest_p=src_dest_p[1]
      $ 545 "FahreAchse"
      $ 546 "stn3_top_hlp_p" "breakAfter"
      set_tcp(p[-3.0E-4,2.5E-4,0.1575,0.0,0.0,0.0])
      movej(get_inverse_kin(pose_trans(stn3_plane, pose_trans(p[.103513391500, -.760903866624, .250613495596, .000363058783, .000522680433, -.002816727210], stn3_top_hlp_p_p)), qnear=stn3_top_hlp_p_q), a=1.7453292519943295, v=1.3962634015954636, r=0.02)
      $ 547 "stn3_home_p" "breakAfter"
      set_tcp(p[-3.0E-4,2.5E-4,0.1575,0.0,0.0,0.0])
      movej(get_inverse_kin(pose_trans(stn3_plane, pose_trans(p[.103513391500, -.760903866624, .250613495596, .000363058783, .000522680433, -.002816727210], stn3_home_p_p)), qnear=stn3_home_p_q), a=2.792526803190927, v=1.7453292519943295, r=0.05)
      $ 548 "FahreAchse"
      $ 549 "stn11_home_p" "breakAfter"
      set_tcp(p[-3.0E-4,2.5E-4,0.1575,0.0,0.0,0.0])
      movej(get_inverse_kin(pose_trans(stn6_plane, pose_trans(p[.776557109756, -.878329076792, .250244777977, -.001605684562, .009314448336, 1.565629725105], stn11_home_p_p)), qnear=stn11_home_p_q), a=1.3962634015954636, v=1.0471975511965976, r=0.05)
      $ 550 "stn11_hlp_p" "breakAfter"
      set_tcp(p[-3.0E-4,2.5E-4,0.1575,0.0,0.0,0.0])
      movej(get_inverse_kin(pose_trans(stn6_plane, pose_trans(p[.776557109756, -.878329076792, .250244777977, -.001605684562, .009314448336, 1.565629725105], stn11_hlp_p_p)), qnear=stn11_hlp_p_q), a=1.3962634015954636, v=1.0471975511965976, r=0.05)
      $ 551 "dest_p" "breakAfter"
      set_tcp(p[-3.0E-4,2.5E-4,0.1575,0.0,0.0,0.0])
      movej(pose_trans(stn6_plane, dest_p), a=1.3962634015954636, v=1.0471975511965976)
      $ 552 "cur_pose≔pose_trans(pose_inv(stn6_plane), get_actual_tcp_pose())"
      global cur_pose= pose_trans ( pose_inv (stn6_plane),  get_actual_tcp_pose ())
      $ 554 "stn11_place_p≔pose_trans(cur_pose, p[0,0,stn11_place_z/1000,0,0,0])"
      global stn11_place_p= pose_trans (cur_pose, p[0,0,stn11_place_z/1000,0,0,0])
      $ 555 "FahreLinear"
      $ 556 "stn11_place_p" "breakAfter"
      set_tcp(p[-3.0E-4,2.5E-4,0.1575,0.0,0.0,0.0])
      movel(pose_trans(stn6_plane, stn11_place_p), a=0.2, v=0.05)
      # begin: URCap Program Node
      #   Source: Robotiq_Grippers, 1.8.13.22852, Robotiq Inc.
      #   Type: Greifer
      $ 557 "Greiferbewegung50% (1)"
      if not(gripper_connected[0]):
        popup("Greifer 1 muss verbunden sein, um dieses Programm auszuführen.", "Keine Verbindung", False, True, True)
      end
      if not(rq_is_gripper_activated("1")):
        popup("Greifer 1 ist nicht aktiviert. Wechseln Sie zur Registerkarte Installation > Greifer, um ihn zu aktivieren und das Programm erneut auszuführen.", "Nicht aktiviert", False, True, True)
      end
      rq_set_pos_spd_for(128, 128, 0, "1")
      rq_wait_pos_spe_for_request(128, 128, 0, "1")
      rq_go_to("1")
      rq_wait("1")
      # end: URCap Program Node
      $ 558 "FahreLinear"
      $ 559 "dest_p" "breakAfter"
      set_tcp(p[-3.0E-4,2.5E-4,0.1575,0.0,0.0,0.0])
      movel(pose_trans(stn6_plane, dest_p), a=1.2, v=0.25)
      # begin: URCap Program Node
      #   Source: Robotiq_Grippers, 1.8.13.22852, Robotiq Inc.
      #   Type: Greifer
      $ 560 "Greifer geschlossen (1)"
      if not(gripper_connected[0]):
        popup("Greifer 1 muss verbunden sein, um dieses Programm auszuführen.", "Keine Verbindung", False, True, True)
      end
      if not(rq_is_gripper_activated("1")):
        popup("Greifer 1 ist nicht aktiviert. Wechseln Sie zur Registerkarte Installation > Greifer, um ihn zu aktivieren und das Programm erneut auszuführen.", "Nicht aktiviert", False, True, True)
      end
      rq_set_pos_spd_for(255, 255, 255, "1")
      rq_wait_pos_spe_for_request(255, 255, 255, "1")
      rq_go_to("1")
      rq_wait("1")
      # end: URCap Program Node
      $ 561 "FahreAchse"
      $ 562 "stn11_hlp_p" "breakAfter"
      set_tcp(p[-3.0E-4,2.5E-4,0.1575,0.0,0.0,0.0])
      movej(get_inverse_kin(pose_trans(stn6_plane, pose_trans(p[.776557109756, -.878329076792, .250244777977, -.001605684562, .009314448336, 1.565629725105], stn11_hlp_p_p)), qnear=stn11_hlp_p_q), a=1.3962634015954636, v=1.0471975511965976, r=0.05)
      $ 563 "stn11_home_p" "breakAfter"
      set_tcp(p[-3.0E-4,2.5E-4,0.1575,0.0,0.0,0.0])
      movej(get_inverse_kin(pose_trans(stn6_plane, pose_trans(p[.776557109756, -.878329076792, .250244777977, -.001605684562, .009314448336, 1.565629725105], stn11_home_p_p)), qnear=stn11_home_p_q), a=1.3962634015954636, v=1.0471975511965976, r=0.05)
      $ 564 "FahreAchse"
      $ 565 "stn3_home_p" "breakAfter"
      set_tcp(p[-3.0E-4,2.5E-4,0.1575,0.0,0.0,0.0])
      movej(get_inverse_kin(pose_trans(stn3_plane, pose_trans(p[.103513391500, -.760903866624, .250613495596, .000363058783, .000522680433, -.002816727210], stn3_home_p_p)), qnear=stn3_home_p_q), a=1.3962634015954636, v=1.0471975511965976)
      $ 566 "Aufruf reset_jobs"
      reset_jobs()
    elif (33 == switch_1):
      $ 567 "Case 33"
      $ 568 "Aufruf stn3_press_run"
      stn3_press_run()
      $ 574 "qMast.set_runtime_alarm(3)"
      qMast.set_runtime_alarm(3)
      $ 575 "FahreAchse"
      $ 576 "stn3_home_p" "breakAfter"
      set_tcp(p[-3.0E-4,2.5E-4,0.1575,0.0,0.0,0.0])
      movej(get_inverse_kin(pose_trans(stn3_plane, pose_trans(p[.103513391500, -.760903866624, .250613495596, .000363058783, .000522680433, -.002816727210], stn3_home_p_p)), qnear=stn3_home_p_q), a=1.3962634015954636, v=1.0471975511965976)
      $ 577 "FahreAchse"
      $ 578 "stn3_pen_pk_u_p" "breakAfter"
      set_tcp(p[-3.0E-4,2.5E-4,0.1575,0.0,0.0,0.0])
      movej(get_inverse_kin(pose_trans(stn6_plane, pose_trans(p[.776557109756, -.878329076792, .250244777977, -.001605684562, .009314448336, 1.565629725105], stn3_pen_pk_u_p_p)), qnear=stn3_pen_pk_u_p_q), a=1.3962634015954636, v=1.0471975511965976)
      $ 579 "FahreLinear"
      $ 580 "stn3_pen_pk_p" "breakAfter"
      set_tcp(p[-3.0E-4,2.5E-4,0.1575,0.0,0.0,0.0])
      movel(pose_trans(stn6_plane, pose_trans(p[.776557109756, -.878329076792, .250244777977, -.001605684562, .009314448336, 1.565629725105], stn3_pen_pk_p_p)), a=1.2, v=0.25)
      # begin: URCap Program Node
      #   Source: Robotiq_Grippers, 1.8.13.22852, Robotiq Inc.
      #   Type: Greifer
      $ 581 "Greiferbewegung50% (1)"
      if not(gripper_connected[0]):
        popup("Greifer 1 muss verbunden sein, um dieses Programm auszuführen.", "Keine Verbindung", False, True, True)
      end
      if not(rq_is_gripper_activated("1")):
        popup("Greifer 1 ist nicht aktiviert. Wechseln Sie zur Registerkarte Installation > Greifer, um ihn zu aktivieren und das Programm erneut auszuführen.", "Nicht aktiviert", False, True, True)
      end
      rq_set_pos_spd_for(128, 255, 128, "1")
      rq_wait_pos_spe_for_request(128, 255, 128, "1")
      rq_go_to("1")
      rq_wait("1")
      # end: URCap Program Node
      $ 582 "stn3_pen_pk_u_p" "breakAfter"
      set_tcp(p[-3.0E-4,2.5E-4,0.1575,0.0,0.0,0.0])
      movel(pose_trans(stn6_plane, pose_trans(p[.776557109756, -.878329076792, .250244777977, -.001605684562, .009314448336, 1.565629725105], stn3_pen_pk_u_p_p)), a=1.2, v=0.25)
      # begin: URCap Program Node
      #   Source: Robotiq_Grippers, 1.8.13.22852, Robotiq Inc.
      #   Type: Greifer
      $ 583 "Greifer geschlossen (1)"
      if not(gripper_connected[0]):
        popup("Greifer 1 muss verbunden sein, um dieses Programm auszuführen.", "Keine Verbindung", False, True, True)
      end
      if not(rq_is_gripper_activated("1")):
        popup("Greifer 1 ist nicht aktiviert. Wechseln Sie zur Registerkarte Installation > Greifer, um ihn zu aktivieren und das Programm erneut auszuführen.", "Nicht aktiviert", False, True, True)
      end
      rq_set_pos_spd_for(255, 255, 128, "1")
      rq_wait_pos_spe_for_request(255, 255, 128, "1")
      rq_go_to("1")
      rq_wait("1")
      # end: URCap Program Node
      $ 584 "FahreAchse"
      $ 585 "stn3_home_p" "breakAfter"
      set_tcp(p[-3.0E-4,2.5E-4,0.1575,0.0,0.0,0.0])
      movej(get_inverse_kin(pose_trans(stn3_plane, pose_trans(p[.103513391500, -.760903866624, .250613495596, .000363058783, .000522680433, -.002816727210], stn3_home_p_p)), qnear=stn3_home_p_q), a=1.3962634015954636, v=1.0471975511965976)
      $ 586 "Aufruf reset_jobs"
      reset_jobs()
    elif (34 == switch_1):
      $ 587 "Case 34"
      $ 588 "Aufruf stn3_press_run"
      stn3_press_run()
      $ 589 "FahreAchse"
      $ 590 "stn3_home_p" "breakAfter"
      set_tcp(p[-3.0E-4,2.5E-4,0.1575,0.0,0.0,0.0])
      movej(get_inverse_kin(pose_trans(stn3_plane, pose_trans(p[.103513391500, -.760903866624, .250613495596, .000363058783, .000522680433, -.002816727210], stn3_home_p_p)), qnear=stn3_home_p_q), a=1.3962634015954636, v=1.0471975511965976)
      $ 591 "FahreAchse"
      $ 592 "stn3_pen_pk_u_p" "breakAfter"
      set_tcp(p[-3.0E-4,2.5E-4,0.1575,0.0,0.0,0.0])
      movej(get_inverse_kin(pose_trans(stn6_plane, pose_trans(p[.776557109756, -.878329076792, .250244777977, -.001605684562, .009314448336, 1.565629725105], stn3_pen_pk_u_p_p)), qnear=stn3_pen_pk_u_p_q), a=1.3962634015954636, v=1.0471975511965976)
      $ 593 "FahreLinear"
      $ 594 "stn3_pen_pk_p" "breakAfter"
      set_tcp(p[-3.0E-4,2.5E-4,0.1575,0.0,0.0,0.0])
      movel(pose_trans(stn6_plane, pose_trans(p[.776557109756, -.878329076792, .250244777977, -.001605684562, .009314448336, 1.565629725105], stn3_pen_pk_p_p)), a=1.2, v=0.25)
      # begin: URCap Program Node
      #   Source: Robotiq_Grippers, 1.8.13.22852, Robotiq Inc.
      #   Type: Greifer
      $ 595 "Greiferbewegung50% (1)"
      if not(gripper_connected[0]):
        popup("Greifer 1 muss verbunden sein, um dieses Programm auszuführen.", "Keine Verbindung", False, True, True)
      end
      if not(rq_is_gripper_activated("1")):
        popup("Greifer 1 ist nicht aktiviert. Wechseln Sie zur Registerkarte Installation > Greifer, um ihn zu aktivieren und das Programm erneut auszuführen.", "Nicht aktiviert", False, True, True)
      end
      rq_set_pos_spd_for(128, 255, 128, "1")
      rq_wait_pos_spe_for_request(128, 255, 128, "1")
      rq_go_to("1")
      rq_wait("1")
      # end: URCap Program Node
      $ 596 "stn3_pen_pk_u_p" "breakAfter"
      set_tcp(p[-3.0E-4,2.5E-4,0.1575,0.0,0.0,0.0])
      movel(pose_trans(stn6_plane, pose_trans(p[.776557109756, -.878329076792, .250244777977, -.001605684562, .009314448336, 1.565629725105], stn3_pen_pk_u_p_p)), a=1.2, v=0.25)
      # begin: URCap Program Node
      #   Source: Robotiq_Grippers, 1.8.13.22852, Robotiq Inc.
      #   Type: Greifer
      $ 597 "Greifer geschlossen (1)"
      if not(gripper_connected[0]):
        popup("Greifer 1 muss verbunden sein, um dieses Programm auszuführen.", "Keine Verbindung", False, True, True)
      end
      if not(rq_is_gripper_activated("1")):
        popup("Greifer 1 ist nicht aktiviert. Wechseln Sie zur Registerkarte Installation > Greifer, um ihn zu aktivieren und das Programm erneut auszuführen.", "Nicht aktiviert", False, True, True)
      end
      rq_set_pos_spd_for(255, 255, 128, "1")
      rq_wait_pos_spe_for_request(255, 255, 128, "1")
      rq_go_to("1")
      rq_wait("1")
      # end: URCap Program Node
      $ 598 "FahreAchse"
      $ 599 "stn3_home_p" "breakAfter"
      set_tcp(p[-3.0E-4,2.5E-4,0.1575,0.0,0.0,0.0])
      movej(get_inverse_kin(pose_trans(stn3_plane, pose_trans(p[.103513391500, -.760903866624, .250613495596, .000363058783, .000522680433, -.002816727210], stn3_home_p_p)), qnear=stn3_home_p_q), a=1.3962634015954636, v=1.0471975511965976)
      $ 600 "Aufruf reset_jobs"
      reset_jobs()
    elif (35 == switch_1):
      $ 601 "Case 35"
      $ 602 "If Test ≟  True "
      if (Test  ==    True  ):
        $ 603 "qMast.set_init_alarm(3)"
        qMast.set_init_alarm(3)
      else:
        $ 604 "Else" "noBreak"
        $ 605 "Aufruf stn3_init_stndby"
        stn3_init_stndby()
        $ 606 "qMast.set_init_alarm(3)"
        qMast.set_init_alarm(3)
        $ 607 "FahreAchse"
        $ 608 "stn3_home_p" "breakAfter"
        set_tcp(p[-3.0E-4,2.5E-4,0.1575,0.0,0.0,0.0])
        movej(get_inverse_kin(pose_trans(stn3_plane, pose_trans(p[.103513391500, -.760903866624, .250613495596, .000363058783, .000522680433, -.002816727210], stn3_home_p_p)), qnear=stn3_home_p_q), a=1.3962634015954636, v=1.0471975511965976)
      end
      $ 609 "Aufruf reset_jobs"
      reset_jobs()
    elif (51 == switch_1):
      $ 610 "Case 51"
      $ 611 "dest_jobID≔jobArr[1]"
      global dest_jobID=jobArr[1]
      $ 612 "FahreAchse"
      $ 613 "stn6_home_p" "breakAfter"
      set_tcp(p[-3.0E-4,2.5E-4,0.1575,0.0,0.0,0.0])
      movej(get_inverse_kin(pose_trans(stn6_plane, pose_trans(p[.776557109756, -.878329076792, .250244777977, -.001605684562, .009314448336, 1.565629725105], stn6_home_p_p)), qnear=stn6_home_p_q), a=2.0943951023931953, v=1.3962634015954636)
      $ 614 "Switch dest_jobID"
      switch_2 = dest_jobID
      $ 615 "Case 41"
      if (41 == switch_2):
        $ 616 "src_dest_p≔qMast.get_loc()"
        global src_dest_p=qMast.get_loc()
        $ 617 "source_p≔src_dest_p[0]"
        global source_p=src_dest_p[0]
        $ 618 "FahreAchse"
        $ 619 "source_p" "breakAfter"
        set_tcp(p[-3.0E-4,2.5E-4,0.1575,0.0,0.0,0.0])
        movej(pose_trans(stn5_plane, source_p), a=1.3962634015954636, v=1.0471975511965976)
        $ 620 "FahreLinear"
        # begin: URCap Program Node
        #   Source: Robotiq_Grippers, 1.8.13.22852, Robotiq Inc.
        #   Type: Greifer
        $ 621 "Greiferbewegung50% (1)"
        if not(gripper_connected[0]):
          popup("Greifer 1 muss verbunden sein, um dieses Programm auszuführen.", "Keine Verbindung", False, True, True)
        end
        if not(rq_is_gripper_activated("1")):
          popup("Greifer 1 ist nicht aktiviert. Wechseln Sie zur Registerkarte Installation > Greifer, um ihn zu aktivieren und das Programm erneut auszuführen.", "Nicht aktiviert", False, True, True)
        end
        rq_set_pos_spd_for(128, 255, 255, "1")
        rq_wait_pos_spe_for_request(128, 255, 255, "1")
        rq_go_to("1")
        rq_wait("1")
        # end: URCap Program Node
        $ 622 "cur_pose≔pose_trans(pose_inv(stn5_plane), get_actual_tcp_pose())"
        global cur_pose= pose_trans ( pose_inv (stn5_plane),  get_actual_tcp_pose ())
        $ 624 "stn5_pick_z_p≔pose_trans(cur_pose, p[0,0,stn5_pick_tb_z/1000,0,0,0])"
        global stn5_pick_z_p= pose_trans (cur_pose, p[0,0,stn5_pick_tb_z/1000,0,0,0])
        $ 625 "stn5_pick_z_p" "breakAfter"
        set_tcp(p[-3.0E-4,2.5E-4,0.1575,0.0,0.0,0.0])
        movel(pose_trans(stn5_plane, stn5_pick_z_p), a=0.25, v=0.1)
        # begin: URCap Program Node
        #   Source: Robotiq_Grippers, 1.8.13.22852, Robotiq Inc.
        #   Type: Greifer
        $ 626 "Greifer geschlossen (1)"
        if not(gripper_connected[0]):
          popup("Greifer 1 muss verbunden sein, um dieses Programm auszuführen.", "Keine Verbindung", False, True, True)
        end
        if not(rq_is_gripper_activated("1")):
          popup("Greifer 1 ist nicht aktiviert. Wechseln Sie zur Registerkarte Installation > Greifer, um ihn zu aktivieren und das Programm erneut auszuführen.", "Nicht aktiviert", False, True, True)
        end
        rq_set_pos_spd_for(255, 128, 128, "1")
        rq_wait_pos_spe_for_request(255, 128, 128, "1")
        rq_go_to("1")
        rq_wait("1")
        # end: URCap Program Node
        $ 627 "source_p" "breakAfter"
        set_tcp(p[-3.0E-4,2.5E-4,0.1575,0.0,0.0,0.0])
        movel(pose_trans(stn5_plane, source_p), a=0.25, v=0.1, r=0.02)
        $ 628 "FahreAchse"
        $ 629 "stn5_stn4_hlp_p" "breakAfter"
        set_tcp(p[-3.0E-4,2.5E-4,0.1575,0.0,0.0,0.0])
        movej(get_inverse_kin(pose_trans(stn6_plane, pose_trans(p[.776557109756, -.878329076792, .250244777977, -.001605684562, .009314448336, 1.565629725105], stn5_stn4_hlp_p_p)), qnear=stn5_stn4_hlp_p_q), a=1.3962634015954636, v=1.0471975511965976, r=0.05)
        $ 630 "Aufruf stn9_decap"
        stn9_decap()
        $ 631 "Aufruf stn4_grab_loop_after"
        stn4_grab_loop_after()
        $ 634 "dest2_jobID≔qMast.stn4_get_next_after(stn4_tube_ok)"
        global dest2_jobID=qMast.stn4_get_next_after(stn4_tube_ok)
        $ 635 "src_dest_p≔qMast.get_loc()"
        global src_dest_p=qMast.get_loc()
        $ 636 "dest_p≔src_dest_p[0]"
        global dest_p=src_dest_p[0]
        $ 637 "Switch dest2_jobID"
        switch_3 = dest2_jobID
        $ 638 "Case 32"
        if (32 == switch_3):
          $ 639 "FahreAchse"
          $ 640 "stn3_home_p" "breakAfter"
          set_tcp(p[-3.0E-4,2.5E-4,0.1575,0.0,0.0,0.0])
          movej(get_inverse_kin(pose_trans(stn3_plane, pose_trans(p[.103513391500, -.760903866624, .250613495596, .000363058783, .000522680433, -.002816727210], stn3_home_p_p)), qnear=stn3_home_p_q), a=1.3962634015954636, v=1.0471975511965976, r=0.1)
          $ 641 "stn3_top_hlp_p" "breakAfter"
          set_tcp(p[-3.0E-4,2.5E-4,0.1575,0.0,0.0,0.0])
          movej(get_inverse_kin(pose_trans(stn3_plane, pose_trans(p[.103513391500, -.760903866624, .250613495596, .000363058783, .000522680433, -.002816727210], stn3_top_hlp_p_p)), qnear=stn3_top_hlp_p_q), a=1.3962634015954636, v=1.0471975511965976, r=0.02)
          $ 642 "dest_p" "breakAfter"
          set_tcp(p[-3.0E-4,2.5E-4,0.1575,0.0,0.0,0.0])
          movej(pose_trans(stn3_plane, dest_p), a=1.3962634015954636, v=1.0471975511965976)
          $ 643 "FahreLinear"
          $ 644 "cur_pose≔pose_trans(pose_inv(stn3_plane), get_actual_tcp_pose())"
          global cur_pose= pose_trans ( pose_inv (stn3_plane),  get_actual_tcp_pose ())
          $ 645 "stn3_rot_set_p≔pose_trans(cur_pose,p[0,0,stn3_rot_z/1000,0,0,0])"
          global stn3_rot_set_p= pose_trans (cur_pose,p[0,0,stn3_rot_z/1000,0,0,0])
          $ 646 "stn3_rot_set_p" "breakAfter"
          set_tcp(p[-3.0E-4,2.5E-4,0.1575,0.0,0.0,0.0])
          movel(pose_trans(stn3_plane, stn3_rot_set_p), a=0.1, v=0.05)
          $ 647 "FahreLinear"
          $ 648 "stn3_rot_angle≔stn4_tube_angle"
          global stn3_rot_angle=stn4_tube_angle
          $ 649 "cur_pose≔pose_trans(pose_inv(stn3_plane), get_actual_tcp_pose())"
          global cur_pose= pose_trans ( pose_inv (stn3_plane),  get_actual_tcp_pose ())
          $ 650 "stn3_rot_p≔pose_trans(cur_pose, p[0,0,0,0,0,d2r(stn3_rot_angle)])"
          global stn3_rot_p= pose_trans (cur_pose, p[0,0,0,0,0,d2r(stn3_rot_angle)])
          $ 651 "stn3_rot_p" "breakAfter"
          set_tcp(p[-3.0E-4,2.5E-4,0.1575,0.0,0.0,0.0])
          movel(pose_trans(stn3_plane, stn3_rot_p), a=0.6, v=0.15)
          $ 652 "FahreLinear"
          $ 653 "cur_pose≔pose_trans(pose_inv(stn3_plane), get_actual_tcp_pose())"
          global cur_pose= pose_trans ( pose_inv (stn3_plane),  get_actual_tcp_pose ())
          $ 654 "stn3_place_z_p≔pose_trans(cur_pose,p[0,0,stn3_place_z/1000,0,0,0])"
          global stn3_place_z_p= pose_trans (cur_pose,p[0,0,stn3_place_z/1000,0,0,0])
          $ 655 "stn3_place_z_p" "breakAfter"
          set_tcp(p[-3.0E-4,2.5E-4,0.1575,0.0,0.0,0.0])
          movel(pose_trans(stn3_plane, stn3_place_z_p), a=0.2, v=0.05)
          # begin: URCap Program Node
          #   Source: Robotiq_Grippers, 1.8.13.22852, Robotiq Inc.
          #   Type: Greifer
          $ 656 "Greiferbewegung50% (1)"
          if not(gripper_connected[0]):
            popup("Greifer 1 muss verbunden sein, um dieses Programm auszuführen.", "Keine Verbindung", False, True, True)
          end
          if not(rq_is_gripper_activated("1")):
            popup("Greifer 1 ist nicht aktiviert. Wechseln Sie zur Registerkarte Installation > Greifer, um ihn zu aktivieren und das Programm erneut auszuführen.", "Nicht aktiviert", False, True, True)
          end
          rq_set_pos_spd_for(128, 64, 255, "1")
          rq_wait_pos_spe_for_request(128, 64, 255, "1")
          rq_go_to("1")
          rq_wait("1")
          # end: URCap Program Node
          $ 657 "FahreLinear"
          $ 658 "cur_pose≔pose_trans(pose_inv(stn3_plane), get_actual_tcp_pose())"
          global cur_pose= pose_trans ( pose_inv (stn3_plane),  get_actual_tcp_pose ())
          $ 659 "stn3_place_z_p≔pose_trans(cur_pose,p[0,0,-stn3_place_z/1000,0,0,0])"
          global stn3_place_z_p= pose_trans (cur_pose,p[0,0,-stn3_place_z/1000,0,0,0])
          $ 660 "stn3_place_z_p" "breakAfter"
          set_tcp(p[-3.0E-4,2.5E-4,0.1575,0.0,0.0,0.0])
          movel(pose_trans(stn3_plane, stn3_place_z_p), a=0.2, v=0.05)
          $ 663 "FahreAchse"
          $ 664 "stn3_top_hlp_p" "breakAfter"
          set_tcp(p[-3.0E-4,2.5E-4,0.1575,0.0,0.0,0.0])
          movej(get_inverse_kin(pose_trans(stn3_plane, pose_trans(p[.103513391500, -.760903866624, .250613495596, .000363058783, .000522680433, -.002816727210], stn3_top_hlp_p_p)), qnear=stn3_top_hlp_p_q), a=1.3962634015954636, v=1.0471975511965976, r=0.02)
          $ 665 "stn3_home_p" "breakAfter"
          set_tcp(p[-3.0E-4,2.5E-4,0.1575,0.0,0.0,0.0])
          movej(get_inverse_kin(pose_trans(stn3_plane, pose_trans(p[.103513391500, -.760903866624, .250613495596, .000363058783, .000522680433, -.002816727210], stn3_home_p_p)), qnear=stn3_home_p_q), a=1.3962634015954636, v=1.0471975511965976)
          # begin: URCap Program Node
          #   Source: Robotiq_Grippers, 1.8.13.22852, Robotiq Inc.
          #   Type: Greifer
          $ 666 "Greifer geschlossen (1)"
          if not(gripper_connected[0]):
            popup("Greifer 1 muss verbunden sein, um dieses Programm auszuführen.", "Keine Verbindung", False, True, True)
          end
          if not(rq_is_gripper_activated("1")):
            popup("Greifer 1 ist nicht aktiviert. Wechseln Sie zur Registerkarte Installation > Greifer, um ihn zu aktivieren und das Programm erneut auszuführen.", "Nicht aktiviert", False, True, True)
          end
          rq_set_pos_spd_for(255, 255, 0, "1")
          rq_wait_pos_spe_for_request(255, 255, 0, "1")
          rq_go_to("1")
          rq_wait("1")
          # end: URCap Program Node
          $ 667 "Aufruf reset_jobs"
          reset_jobs()
        elif (102 == switch_3):
          $ 668 "Case 102"
          $ 669 "FahreAchse"
          $ 670 "stn10_hlp_p" "breakAfter"
          set_tcp(p[-3.0E-4,2.5E-4,0.1575,0.0,0.0,0.0])
          movej(get_inverse_kin(pose_trans(stn6_plane, pose_trans(p[.779413821965, -.869656427631, .149271774994, -.000554336510, .003016566406, 1.568064465904], stn10_hlp_p_p)), qnear=stn10_hlp_p_q), a=1.3962634015954636, v=1.0471975511965976)
          $ 671 "FahreLinear"
          $ 672 "dest_p" "breakAfter"
          set_tcp(p[-3.0E-4,2.5E-4,0.1575,0.0,0.0,0.0])
          movel(pose_trans(stn6_plane, dest_p), a=1.2, v=0.25)
          $ 673 "cur_pose≔pose_trans(pose_inv(stn6_plane), get_actual_tcp_pose())"
          global cur_pose= pose_trans ( pose_inv (stn6_plane),  get_actual_tcp_pose ())
          $ 674 "stn10_place_p≔pose_trans(cur_pose, p[0,0,stn10_place_z/1000,0,0,0])"
          global stn10_place_p= pose_trans (cur_pose, p[0,0,stn10_place_z/1000,0,0,0])
          $ 675 "FahreLinear"
          $ 676 "stn10_place_p" "breakAfter"
          set_tcp(p[-3.0E-4,2.5E-4,0.1575,0.0,0.0,0.0])
          movel(pose_trans(stn6_plane, stn10_place_p), a=0.2, v=0.075)
          # begin: URCap Program Node
          #   Source: Robotiq_Grippers, 1.8.13.22852, Robotiq Inc.
          #   Type: Greifer
          $ 677 "Greiferbewegung50% (1)"
          if not(gripper_connected[0]):
            popup("Greifer 1 muss verbunden sein, um dieses Programm auszuführen.", "Keine Verbindung", False, True, True)
          end
          if not(rq_is_gripper_activated("1")):
            popup("Greifer 1 ist nicht aktiviert. Wechseln Sie zur Registerkarte Installation > Greifer, um ihn zu aktivieren und das Programm erneut auszuführen.", "Nicht aktiviert", False, True, True)
          end
          rq_set_pos_spd_for(128, 255, 0, "1")
          rq_wait_pos_spe_for_request(128, 255, 0, "1")
          rq_go_to("1")
          rq_wait("1")
          # end: URCap Program Node
          $ 678 "dest_p" "breakAfter"
          set_tcp(p[-3.0E-4,2.5E-4,0.1575,0.0,0.0,0.0])
          movel(pose_trans(stn6_plane, dest_p), a=1.2, v=0.25)
          # begin: URCap Program Node
          #   Source: Robotiq_Grippers, 1.8.13.22852, Robotiq Inc.
          #   Type: Greifer
          $ 679 "Greifer geschlossen (1)"
          if not(gripper_connected[0]):
            popup("Greifer 1 muss verbunden sein, um dieses Programm auszuführen.", "Keine Verbindung", False, True, True)
          end
          if not(rq_is_gripper_activated("1")):
            popup("Greifer 1 ist nicht aktiviert. Wechseln Sie zur Registerkarte Installation > Greifer, um ihn zu aktivieren und das Programm erneut auszuführen.", "Nicht aktiviert", False, True, True)
          end
          rq_set_pos_spd_for(255, 255, 255, "1")
          rq_wait_pos_spe_for_request(255, 255, 255, "1")
          rq_go_to("1")
          rq_wait("1")
          # end: URCap Program Node
          $ 680 "FahreAchse"
          $ 681 "stn10_hlp_p" "breakAfter"
          set_tcp(p[-3.0E-4,2.5E-4,0.1575,0.0,0.0,0.0])
          movej(get_inverse_kin(pose_trans(stn6_plane, pose_trans(p[.779413821965, -.869656427631, .149271774994, -.000554336510, .003016566406, 1.568064465904], stn10_hlp_p_p)), qnear=stn10_hlp_p_q), a=1.3962634015954636, v=1.0471975511965976, r=0.1)
          $ 682 "stn6_home_p" "breakAfter"
          set_tcp(p[-3.0E-4,2.5E-4,0.1575,0.0,0.0,0.0])
          movej(get_inverse_kin(pose_trans(stn6_plane, pose_trans(p[.776557109756, -.878329076792, .250244777977, -.001605684562, .009314448336, 1.565629725105], stn6_home_p_p)), qnear=stn6_home_p_q), a=1.3962634015954636, v=1.0471975511965976)
          $ 683 "Aufruf reset_jobs"
          reset_jobs()
        elif (143 == switch_3):
          $ 684 "Case 143"
          $ 685 "FahreAchse"
          $ 686 "dest_p" "breakAfter"
          set_tcp(p[-3.0E-4,2.5E-4,0.1575,0.0,0.0,0.0])
          movej(pose_trans(stn6_plane, dest_p), a=1.3962634015954636, v=1.0471975511965976)
          $ 687 "FahreLinear"
          $ 688 "cur_pose≔pose_trans(pose_inv(stn6_plane), get_actual_tcp_pose())"
          global cur_pose= pose_trans ( pose_inv (stn6_plane),  get_actual_tcp_pose ())
          $ 689 "stn14_set_rot_p≔pose_trans(cur_pose, p[0,0,stn14_tb_rot_z/1000,0,0,0])"
          global stn14_set_rot_p= pose_trans (cur_pose, p[0,0,stn14_tb_rot_z/1000,0,0,0])
          $ 690 "stn14_set_rot_p" "breakAfter"
          set_tcp(p[-3.0E-4,2.5E-4,0.1575,0.0,0.0,0.0])
          movel(pose_trans(stn6_plane, stn14_set_rot_p), a=0.2, v=0.075)
          $ 691 "cur_pose≔pose_trans(pose_inv(stn6_plane), get_actual_tcp_pose())"
          global cur_pose= pose_trans ( pose_inv (stn6_plane),  get_actual_tcp_pose ())
          $ 692 "stn14_rot_p≔pose_trans(cur_pose, p[0,0,0,0,0,d2r(stn4_tube_angle)])"
          global stn14_rot_p= pose_trans (cur_pose, p[0,0,0,0,0,d2r(stn4_tube_angle)])
          $ 693 "stn14_rot_p" "breakAfter"
          set_tcp(p[-3.0E-4,2.5E-4,0.1575,0.0,0.0,0.0])
          movel(pose_trans(stn6_plane, stn14_rot_p), a=0.5, v=0.1)
          $ 694 "cur_pose≔pose_trans(pose_inv(stn6_plane), get_actual_tcp_pose())"
          global cur_pose= pose_trans ( pose_inv (stn6_plane),  get_actual_tcp_pose ())
          $ 695 "stn14_plac_tb_p≔pose_trans(cur_pose, p[0,0,stn14_tb_pl_z/1000,0,0,0])"
          global stn14_plac_tb_p= pose_trans (cur_pose, p[0,0,stn14_tb_pl_z/1000,0,0,0])
          $ 696 "stn14_plac_tb_p" "breakAfter"
          set_tcp(p[-3.0E-4,2.5E-4,0.1575,0.0,0.0,0.0])
          movel(pose_trans(stn6_plane, stn14_plac_tb_p), a=0.4, v=0.1)
          # begin: URCap Program Node
          #   Source: Robotiq_Grippers, 1.8.13.22852, Robotiq Inc.
          #   Type: Greifer
          $ 697 "Greiferbewegung70% (1)"
          if not(gripper_connected[0]):
            popup("Greifer 1 muss verbunden sein, um dieses Programm auszuführen.", "Keine Verbindung", False, True, True)
          end
          if not(rq_is_gripper_activated("1")):
            popup("Greifer 1 ist nicht aktiviert. Wechseln Sie zur Registerkarte Installation > Greifer, um ihn zu aktivieren und das Programm erneut auszuführen.", "Nicht aktiviert", False, True, True)
          end
          rq_set_pos_spd_for(179, 64, 255, "1")
          rq_wait_pos_spe_for_request(179, 64, 255, "1")
          rq_go_to("1")
          rq_wait("1")
          # end: URCap Program Node
          $ 698 "cur_pose≔pose_trans(pose_inv(stn6_plane), get_actual_tcp_pose())"
          global cur_pose= pose_trans ( pose_inv (stn6_plane),  get_actual_tcp_pose ())
          $ 699 "stn14_plac_tb_p≔pose_trans(cur_pose, p[0,0,-50/1000,0,0,0])"
          global stn14_plac_tb_p= pose_trans (cur_pose, p[0,0,-50/1000,0,0,0])
          $ 700 "stn14_plac_tb_p" "breakAfter"
          set_tcp(p[-3.0E-4,2.5E-4,0.1575,0.0,0.0,0.0])
          movel(pose_trans(stn6_plane, stn14_plac_tb_p), a=0.4, v=0.1)
          $ 701 "FahreAchse"
          $ 702 "stn14_rot_hlp_p" "breakAfter"
          set_tcp(p[-3.0E-4,2.5E-4,0.1575,0.0,0.0,0.0])
          movej(get_inverse_kin(pose_trans(stn6_plane, pose_trans(p[.776557109756, -.878329076792, .250244777977, -.001605684562, .009314448336, 1.565629725105], stn14_rot_hlp_p_p)), qnear=stn14_rot_hlp_p_q), a=2.0943951023931953, v=1.3962634015954636, r=0.05)
          $ 703 "stn6_home_p" "breakAfter"
          set_tcp(p[-3.0E-4,2.5E-4,0.1575,0.0,0.0,0.0])
          movej(get_inverse_kin(pose_trans(stn6_plane, pose_trans(p[.776557109756, -.878329076792, .250244777977, -.001605684562, .009314448336, 1.565629725105], stn6_home_p_p)), qnear=stn6_home_p_q), a=2.0943951023931953, v=1.3962634015954636)
          # begin: URCap Program Node
          #   Source: Robotiq_Grippers, 1.8.13.22852, Robotiq Inc.
          #   Type: Greifer
          $ 704 "Greifer geschlossen (1)"
          if not(gripper_connected[0]):
            popup("Greifer 1 muss verbunden sein, um dieses Programm auszuführen.", "Keine Verbindung", False, True, True)
          end
          if not(rq_is_gripper_activated("1")):
            popup("Greifer 1 ist nicht aktiviert. Wechseln Sie zur Registerkarte Installation > Greifer, um ihn zu aktivieren und das Programm erneut auszuführen.", "Nicht aktiviert", False, True, True)
          end
          rq_set_pos_spd_for(255, 255, 255, "1")
          rq_wait_pos_spe_for_request(255, 255, 255, "1")
          rq_go_to("1")
          rq_wait("1")
          # end: URCap Program Node
          $ 705 "Aufruf reset_jobs"
          reset_jobs()
        end
      elif (55 == switch_2):
        $ 706 "Case 55"
        $ 707 "src_dest_p≔qMast.get_loc()"
        global src_dest_p=qMast.get_loc()
        $ 708 "source_p≔src_dest_p[0]"
        global source_p=src_dest_p[0]
        $ 709 "dest_p≔src_dest_p[1]"
        global dest_p=src_dest_p[1]
        $ 710 "FahreAchse"
        $ 711 "stn5_stn4_hlp_p" "breakAfter"
        set_tcp(p[-3.0E-4,2.5E-4,0.1575,0.0,0.0,0.0])
        movej(get_inverse_kin(pose_trans(stn6_plane, pose_trans(p[.776557109756, -.878329076792, .250244777977, -.001605684562, .009314448336, 1.565629725105], stn5_stn4_hlp_p_p)), qnear=stn5_stn4_hlp_p_q), a=1.3962634015954636, v=1.0471975511965976, r=0.05)
        $ 712 "FahreAchse"
        $ 713 "source_p" "breakAfter"
        set_tcp(p[-3.0E-4,2.5E-4,0.1575,0.0,0.0,0.0])
        movej(pose_trans(stn5_plane, source_p), a=1.3962634015954636, v=1.0471975511965976)
        # begin: URCap Program Node
        #   Source: Robotiq_Grippers, 1.8.13.22852, Robotiq Inc.
        #   Type: Greifer
        $ 714 "Greiferbewegung50% (1)"
        if not(gripper_connected[0]):
          popup("Greifer 1 muss verbunden sein, um dieses Programm auszuführen.", "Keine Verbindung", False, True, True)
        end
        if not(rq_is_gripper_activated("1")):
          popup("Greifer 1 ist nicht aktiviert. Wechseln Sie zur Registerkarte Installation > Greifer, um ihn zu aktivieren und das Programm erneut auszuführen.", "Nicht aktiviert", False, True, True)
        end
        rq_set_pos_spd_for(127, 255, 255, "1")
        rq_wait_pos_spe_for_request(127, 255, 255, "1")
        rq_go_to("1")
        rq_wait("1")
        # end: URCap Program Node
        $ 715 "cur_pose≔pose_trans(pose_inv(stn5_plane), get_actual_tcp_pose())"
        global cur_pose= pose_trans ( pose_inv (stn5_plane),  get_actual_tcp_pose ())
        $ 716 "stn5_cw_pick_p≔pose_trans(cur_pose, p[0,0,stn5_pick_tb_z/1000,0,0,0])"
        global stn5_cw_pick_p= pose_trans (cur_pose, p[0,0,stn5_pick_tb_z/1000,0,0,0])
        $ 717 "FahreLinear"
        $ 718 "stn5_cw_pick_p" "breakAfter"
        set_tcp(p[-3.0E-4,2.5E-4,0.1575,0.0,0.0,0.0])
        movel(pose_trans(stn5_plane, stn5_cw_pick_p), a=0.3, v=0.1)
        # begin: URCap Program Node
        #   Source: Robotiq_Grippers, 1.8.13.22852, Robotiq Inc.
        #   Type: Greifer
        $ 719 "Greifer geschlossen (1)"
        if not(gripper_connected[0]):
          popup("Greifer 1 muss verbunden sein, um dieses Programm auszuführen.", "Keine Verbindung", False, True, True)
        end
        if not(rq_is_gripper_activated("1")):
          popup("Greifer 1 ist nicht aktiviert. Wechseln Sie zur Registerkarte Installation > Greifer, um ihn zu aktivieren und das Programm erneut auszuführen.", "Nicht aktiviert", False, True, True)
        end
        rq_set_pos_spd_for(255, 128, 128, "1")
        rq_wait_pos_spe_for_request(255, 128, 128, "1")
        rq_go_to("1")
        rq_wait("1")
        # end: URCap Program Node
        $ 720 "source_p" "breakAfter"
        set_tcp(p[-3.0E-4,2.5E-4,0.1575,0.0,0.0,0.0])
        movel(pose_trans(stn5_plane, source_p), a=0.3, v=0.1)
        $ 721 "FahreAchse"
        $ 722 "stn5_stn4_hlp_p" "breakAfter"
        set_tcp(p[-3.0E-4,2.5E-4,0.1575,0.0,0.0,0.0])
        movej(get_inverse_kin(pose_trans(stn6_plane, pose_trans(p[.776557109756, -.878329076792, .250244777977, -.001605684562, .009314448336, 1.565629725105], stn5_stn4_hlp_p_p)), qnear=stn5_stn4_hlp_p_q), a=1.3962634015954636, v=1.0471975511965976, r=0.05)
        $ 723 "FahreAchse"
        $ 724 "dest_p" "breakAfter"
        set_tcp(p[-3.0E-4,2.5E-4,0.1575,0.0,0.0,0.0])
        movej(pose_trans(stn5_plane, dest_p), a=1.3962634015954636, v=1.0471975511965976)
        $ 725 "cur_pose≔pose_trans(pose_inv(stn5_plane), get_actual_tcp_pose())"
        global cur_pose= pose_trans ( pose_inv (stn5_plane),  get_actual_tcp_pose ())
        $ 726 "stn5_cw_place_p≔pose_trans(cur_pose, p[0,0,stn5_place_cw_z/1000,0,0,0])"
        global stn5_cw_place_p= pose_trans (cur_pose, p[0,0,stn5_place_cw_z/1000,0,0,0])
        $ 727 "FahreLinear"
        $ 728 "stn5_cw_place_p" "breakAfter"
        set_tcp(p[-3.0E-4,2.5E-4,0.1575,0.0,0.0,0.0])
        movel(pose_trans(stn5_plane, stn5_cw_place_p), a=0.3, v=0.1)
        # begin: URCap Program Node
        #   Source: Robotiq_Grippers, 1.8.13.22852, Robotiq Inc.
        #   Type: Greifer
        $ 729 "Greiferbewegung60% (1)"
        if not(gripper_connected[0]):
          popup("Greifer 1 muss verbunden sein, um dieses Programm auszuführen.", "Keine Verbindung", False, True, True)
        end
        if not(rq_is_gripper_activated("1")):
          popup("Greifer 1 ist nicht aktiviert. Wechseln Sie zur Registerkarte Installation > Greifer, um ihn zu aktivieren und das Programm erneut auszuführen.", "Nicht aktiviert", False, True, True)
        end
        rq_set_pos_spd_for(153, 255, 0, "1")
        rq_wait_pos_spe_for_request(153, 255, 0, "1")
        rq_go_to("1")
        rq_wait("1")
        # end: URCap Program Node
        $ 730 "dest_p" "breakAfter"
        set_tcp(p[-3.0E-4,2.5E-4,0.1575,0.0,0.0,0.0])
        movel(pose_trans(stn5_plane, dest_p), a=0.3, v=0.1)
        # begin: URCap Program Node
        #   Source: Robotiq_Grippers, 1.8.13.22852, Robotiq Inc.
        #   Type: Greifer
        $ 731 "Greifer geschlossen (1)"
        if not(gripper_connected[0]):
          popup("Greifer 1 muss verbunden sein, um dieses Programm auszuführen.", "Keine Verbindung", False, True, True)
        end
        if not(rq_is_gripper_activated("1")):
          popup("Greifer 1 ist nicht aktiviert. Wechseln Sie zur Registerkarte Installation > Greifer, um ihn zu aktivieren und das Programm erneut auszuführen.", "Nicht aktiviert", False, True, True)
        end
        rq_set_pos_spd_for(255, 255, 0, "1")
        rq_wait_pos_spe_for_request(255, 255, 0, "1")
        rq_go_to("1")
        rq_wait("1")
        # end: URCap Program Node
        $ 732 "FahreAchse"
        $ 733 "stn6_home_p" "breakAfter"
        set_tcp(p[-3.0E-4,2.5E-4,0.1575,0.0,0.0,0.0])
        movej(get_inverse_kin(pose_trans(stn6_plane, pose_trans(p[.776557109756, -.878329076792, .250244777977, -.001605684562, .009314448336, 1.565629725105], stn6_home_p_p)), qnear=stn6_home_p_q), a=1.3962634015954636, v=1.0471975511965976)
        $ 734 "Aufruf reset_jobs"
        reset_jobs()
      elif (62 == switch_2):
        $ 735 "Case 62"
        $ 736 "stn5_dest_4ps_p≔qMast.stn5_get_loc()"
        global stn5_dest_4ps_p=qMast.stn5_get_loc()
        $ 737 "FahreAchse"
        $ 738 "stn6_help_p" "breakAfter"
        set_tcp(p[-3.0E-4,2.5E-4,0.1575,0.0,0.0,0.0])
        movej(get_inverse_kin(pose_trans(stn6_plane, pose_trans(p[.776557109756, -.878329076792, .250244777977, -.001605684562, .009314448336, 1.565629725105], stn6_help_p_p)), qnear=stn6_help_p_q), a=1.3962634015954636, v=1.0471975511965976)
        $ 739 "If Test ≟  True "
        if (Test  ==    True  ):
          $ 740 "qMast.set_runtime_alarm(6)"
          qMast.set_runtime_alarm(6)
        else:
          $ 741 "Else" "noBreak"
          $ 742 "stn6_hatch_open≔qMast.stn6_hatch_open()"
          global stn6_hatch_open=qMast.stn6_hatch_open()
          $ 743 "If stn6_hatch_open ≟  True "
          if (stn6_hatch_open  ==    True  ):
            $ 744 "stn5_loop_count≔0"
            global stn5_loop_count=0
            $ 745 "Schleife 4 mal"
            Loop_2 = 0
            while (Loop_2 < 4):
              $ 746 "FahreAchse"
              $ 747 "stn6_help_p" "breakAfter"
              set_tcp(p[-3.0E-4,2.5E-4,0.1575,0.0,0.0,0.0])
              movej(get_inverse_kin(pose_trans(stn6_plane, pose_trans(p[.776557109756, -.878329076792, .250244777977, -.001605684562, .009314448336, 1.565629725105], stn6_help_p_p)), qnear=stn6_help_p_q), a=1.3962634015954636, v=1.0471975511965976)
              $ 748 "stn6_set_rotor≔qMast.stn6_set_rotor_position(stn5_loop_count + 1)"
              global stn6_set_rotor=qMast.stn6_set_rotor_position(stn5_loop_count + 1)
              $ 749 "If stn6_set_rotor ≟  True "
              if (stn6_set_rotor  ==    True  ):
                $ 750 "stn5_source_p≔stn5_dest_4ps_p[stn5_loop_count]"
                global stn5_source_p=stn5_dest_4ps_p[stn5_loop_count]
                $ 751 "FahreAchse"
                $ 752 "stn5_source_p" "breakAfter"
                set_tcp(p[-3.0E-4,2.5E-4,0.1575,0.0,0.0,0.0])
                movej(pose_trans(stn5_plane, stn5_source_p), a=1.3962634015954636, v=1.0471975511965976)
                $ 753 "FahreLinear"
                # begin: URCap Program Node
                #   Source: Robotiq_Grippers, 1.8.13.22852, Robotiq Inc.
                #   Type: Greifer
                $ 754 "Greiferbewegung50% (1)"
                if not(gripper_connected[0]):
                  popup("Greifer 1 muss verbunden sein, um dieses Programm auszuführen.", "Keine Verbindung", False, True, True)
                end
                if not(rq_is_gripper_activated("1")):
                  popup("Greifer 1 ist nicht aktiviert. Wechseln Sie zur Registerkarte Installation > Greifer, um ihn zu aktivieren und das Programm erneut auszuführen.", "Nicht aktiviert", False, True, True)
                end
                rq_set_pos_spd_for(128, 255, 255, "1")
                rq_wait_pos_spe_for_request(128, 255, 255, "1")
                rq_go_to("1")
                rq_wait("1")
                # end: URCap Program Node
                $ 755 "cur_pose≔pose_trans(pose_inv(stn5_plane), get_actual_tcp_pose())"
                global cur_pose= pose_trans ( pose_inv (stn5_plane),  get_actual_tcp_pose ())
                $ 756 "stn5_pick_rk_p≔pose_trans(cur_pose, p[0,0,stn5_pick_rk_z/1000,0,0,0])"
                global stn5_pick_rk_p= pose_trans (cur_pose, p[0,0,stn5_pick_rk_z/1000,0,0,0])
                $ 757 "stn5_pick_rk_p" "breakAfter"
                set_tcp(p[-3.0E-4,2.5E-4,0.1575,0.0,0.0,0.0])
                movel(pose_trans(stn5_plane, stn5_pick_rk_p), a=0.8, v=0.15)
                # begin: URCap Program Node
                #   Source: Robotiq_Grippers, 1.8.13.22852, Robotiq Inc.
                #   Type: Greifer
                $ 758 "Greifer geschlossen (1)"
                if not(gripper_connected[0]):
                  popup("Greifer 1 muss verbunden sein, um dieses Programm auszuführen.", "Keine Verbindung", False, True, True)
                end
                if not(rq_is_gripper_activated("1")):
                  popup("Greifer 1 ist nicht aktiviert. Wechseln Sie zur Registerkarte Installation > Greifer, um ihn zu aktivieren und das Programm erneut auszuführen.", "Nicht aktiviert", False, True, True)
                end
                rq_set_pos_spd_for(255, 128, 128, "1")
                rq_wait_pos_spe_for_request(255, 128, 128, "1")
                rq_go_to("1")
                rq_wait("1")
                # end: URCap Program Node
                $ 759 "stn5_source_p" "breakAfter"
                set_tcp(p[-3.0E-4,2.5E-4,0.1575,0.0,0.0,0.0])
                movel(pose_trans(stn5_plane, stn5_source_p), a=0.8, v=0.15)
                $ 760 "FahreAchse"
                $ 761 "stn6_help_p" "breakAfter"
                set_tcp(p[-3.0E-4,2.5E-4,0.1575,0.0,0.0,0.0])
                movej(get_inverse_kin(pose_trans(stn6_plane, pose_trans(p[.776557109756, -.878329076792, .250244777977, -.001605684562, .009314448336, 1.565629725105], stn6_help_p_p)), qnear=stn6_help_p_q), a=1.3962634015954636, v=1.0471975511965976, r=0.05)
                $ 762 "stn6_place_p" "breakAfter"
                set_tcp(p[-3.0E-4,2.5E-4,0.1575,0.0,0.0,0.0])
                movej(get_inverse_kin(pose_trans(stn6_plane, pose_trans(p[.776557109756, -.878329076792, .250244777977, -.001605684562, .009314448336, 1.565629725105], stn6_place_p_p)), qnear=stn6_place_p_q), a=1.3962634015954636, v=1.0471975511965976)
                $ 763 "FahreLinear"
                $ 764 "cur_pose≔pose_trans(pose_inv(stn6_plane), get_actual_tcp_pose())"
                global cur_pose= pose_trans ( pose_inv (stn6_plane),  get_actual_tcp_pose ())
                $ 765 "stn6_place_z_p≔pose_trans(cur_pose, p[0,0,stn6_place_z/1000,0,0,0])"
                global stn6_place_z_p= pose_trans (cur_pose, p[0,0,stn6_place_z/1000,0,0,0])
                $ 766 "stn6_place_z_p" "breakAfter"
                set_tcp(p[-3.0E-4,2.5E-4,0.1575,0.0,0.0,0.0])
                movel(pose_trans(stn6_plane, stn6_place_z_p), a=0.3, v=0.075)
                # begin: URCap Program Node
                #   Source: Robotiq_Grippers, 1.8.13.22852, Robotiq Inc.
                #   Type: Greifer
                $ 767 "Greiferbewegung40% (1)"
                if not(gripper_connected[0]):
                  popup("Greifer 1 muss verbunden sein, um dieses Programm auszuführen.", "Keine Verbindung", False, True, True)
                end
                if not(rq_is_gripper_activated("1")):
                  popup("Greifer 1 ist nicht aktiviert. Wechseln Sie zur Registerkarte Installation > Greifer, um ihn zu aktivieren und das Programm erneut auszuführen.", "Nicht aktiviert", False, True, True)
                end
                rq_set_pos_spd_for(102, 255, 0, "1")
                rq_wait_pos_spe_for_request(102, 255, 0, "1")
                rq_go_to("1")
                rq_wait("1")
                # end: URCap Program Node
                $ 768 "FahreLinear"
                $ 769 "stn6_place_p" "breakAfter"
                set_tcp(p[-3.0E-4,2.5E-4,0.1575,0.0,0.0,0.0])
                movel(pose_trans(stn6_plane, pose_trans(p[.776557109756, -.878329076792, .250244777977, -.001605684562, .009314448336, 1.565629725105], stn6_place_p_p)), a=1.2, v=0.25)
                # begin: URCap Program Node
                #   Source: Robotiq_Grippers, 1.8.13.22852, Robotiq Inc.
                #   Type: Greifer
                $ 770 "Greifer geschlossen (1)"
                if not(gripper_connected[0]):
                  popup("Greifer 1 muss verbunden sein, um dieses Programm auszuführen.", "Keine Verbindung", False, True, True)
                end
                if not(rq_is_gripper_activated("1")):
                  popup("Greifer 1 ist nicht aktiviert. Wechseln Sie zur Registerkarte Installation > Greifer, um ihn zu aktivieren und das Programm erneut auszuführen.", "Nicht aktiviert", False, True, True)
                end
                rq_set_pos_spd_for(255, 128, 255, "1")
                rq_wait_pos_spe_for_request(255, 128, 255, "1")
                rq_go_to("1")
                rq_wait("1")
                # end: URCap Program Node
                $ 771 "stn5_loop_count≔stn5_loop_count + 1"
                global stn5_loop_count=stn5_loop_count + 1
              end
              Loop_2 = Loop_2 + 1
            end
          end
          $ 772 "FahreAchse"
          $ 773 "stn6_help_p" "breakAfter"
          set_tcp(p[-3.0E-4,2.5E-4,0.1575,0.0,0.0,0.0])
          movej(get_inverse_kin(pose_trans(stn6_plane, pose_trans(p[.776557109756, -.878329076792, .250244777977, -.001605684562, .009314448336, 1.565629725105], stn6_help_p_p)), qnear=stn6_help_p_q), a=1.3962634015954636, v=1.0471975511965976)
          $ 774 "stn6_hatch_clse≔qMast.stn6_hatch_close()"
          global stn6_hatch_clse=qMast.stn6_hatch_close()
          $ 775 "If stn6_hatch_clse ≟  True "
          if (stn6_hatch_clse  ==    True  ):
            $ 776 "stn6_start_fuge≔qMast.stn6_start_centrifuge()"
            global stn6_start_fuge=qMast.stn6_start_centrifuge()
            $ 777 "qMast.set_runtime_alarm(6)"
            qMast.set_runtime_alarm(6)
          end
        end
        $ 778 "FahreAchse"
        $ 779 "stn6_home_p" "breakAfter"
        set_tcp(p[-3.0E-4,2.5E-4,0.1575,0.0,0.0,0.0])
        movej(get_inverse_kin(pose_trans(stn6_plane, pose_trans(p[.776557109756, -.878329076792, .250244777977, -.001605684562, .009314448336, 1.565629725105], stn6_home_p_p)), qnear=stn6_home_p_q), a=1.3962634015954636, v=1.0471975511965976)
        $ 780 "Aufruf reset_jobs"
        reset_jobs()
      end
    elif (54 == switch_1):
      $ 781 "Case 54"
      $ 782 "dest_jobID≔jobArr[1]"
      global dest_jobID=jobArr[1]
      $ 783 "src_dest_p≔qMast.get_loc()"
      global src_dest_p=qMast.get_loc()
      $ 784 "source_p≔src_dest_p[0]"
      global source_p=src_dest_p[0]
      $ 785 "dest_p≔src_dest_p[1]"
      global dest_p=src_dest_p[1]
      $ 786 "Switch dest_jobID"
      switch_2 = dest_jobID
      $ 787 "Case 52"
      if (52 == switch_2):
        $ 788 "FahreAchse"
        $ 789 "stn6_home_p" "breakAfter"
        set_tcp(p[-3.0E-4,2.5E-4,0.1575,0.0,0.0,0.0])
        movej(get_inverse_kin(pose_trans(stn6_plane, pose_trans(p[.776557109756, -.878329076792, .250244777977, -.001605684562, .009314448336, 1.565629725105], stn6_home_p_p)), qnear=stn6_home_p_q), a=1.3962634015954636, v=1.0471975511965976)
        $ 790 "FahreAchse"
        $ 791 "source_p" "breakAfter"
        set_tcp(p[-3.0E-4,2.5E-4,0.1575,0.0,0.0,0.0])
        movej(pose_trans(stn5_plane, source_p), a=1.3962634015954636, v=1.0471975511965976)
        # begin: URCap Program Node
        #   Source: Robotiq_Grippers, 1.8.13.22852, Robotiq Inc.
        #   Type: Greifer
        $ 792 "Greiferbewegung50% (1)"
        if not(gripper_connected[0]):
          popup("Greifer 1 muss verbunden sein, um dieses Programm auszuführen.", "Keine Verbindung", False, True, True)
        end
        if not(rq_is_gripper_activated("1")):
          popup("Greifer 1 ist nicht aktiviert. Wechseln Sie zur Registerkarte Installation > Greifer, um ihn zu aktivieren und das Programm erneut auszuführen.", "Nicht aktiviert", False, True, True)
        end
